VAR (* inputs/outputs *)

	ResetOld : BOOL;
	KeyResetOld : BOOL;
	AuxResetActivation : BOOL;
	ResetActivation : BOOL;
	Signals : ARRAY[1..256] OF BOOL;		(*each cell represents a signal code, used to know if signal is Active *)
	NumberOfAlarms : INT;			(* Counting processed alarms *)
	NumberOfAnomalies : INT;		(* Counting processed anomalies *)
	NumberOfWarnings : INT;		(* Counting processed warnings *)
	NumberOfInformation : INT;		(* Counting processed information *)
	ActiveSignalCodes : ARRAY[0..256] OF WORD;	(*each cell represents a Counted Active Signal Code, used to distinguish active/inactive in cronological sense*)
	NumberOfActiveAlarms : INT;		(* Counting active alarms *)
	NumberOfActiveAnomalies : INT;		(* Counting active anomalies *)
	NumberOfActiveWarning : INT;		(* Counting active warnings *)
	NumberOfActiveInformation : INT;	(* Counting active information *)
	SignalManagementError : BOOL;		(* not used for now *)
	Index : INT;	                             (*To trace working signal *)
	BaseIndex : INT;			(* To Trace offset depending on signal type *)
	i: INT;		(* Used in Reset Activation FOR Cycle *)
	AutoResetCondition: BOOL;	(* FALSE for Alarms/Anomalies, TRUE for Warning/Info *)
	AuxResetCondition: BOOL;	(* FALSE when AUX_RESET needed, TRUE for others *)
	SignalsCounters : ARRAY [1..256] OF INT;	(* Counters for Provisional Reset Condition *)
	ProvisionFlag: BOOL := FALSE;

END_VAR
CASE OperationType OF

	INIT: (* INIT PHASE *)			(* Reset Arrays - 1 Time*)

		IF KeyReset THEN

			FOR i:=1 TO 256 DO
				Signals[i] := FALSE;
				ActiveSignalCodes[i] := 0;		(* =NONE *)
				SignalsCounters[i] := 0;
			END_FOR

		END_IF

	START_CONFIGURATION: (* START_CONFIGURATION *)			(* Reset Alarms Count 1-Time *)

		NumberOfAlarms := 0;
		NumberOfAnomalies := 0;
		NumberOfWarnings := 0;
		NumberOfInformation := 0;

	CONFIGURATION:  (* CONFIGURATION PHASE*)					(* counting signals - Cycle over all possible signals *)

		CASE (WORD_TO_INT(SignalType AND SIGNAL_TYPE_MASK)) OF
			1:   (*ALARMS*)

				NumberOfAlarms := NumberOfAlarms + 1;

			2:   (*ANOMALIES*)

				NumberOfAnomalies := NumberOfAnomalies + 1;

			3:  (*WARNINGS*)

				NumberOfWarnings := NumberOfWarnings + 1;

			4:  (*INFORMATIONS*)

				NumberOfInformation := NumberOfInformation + 1;

		END_CASE

	START_GENERATION:  (* START GENERATION PHASE*)			(* Prepare for generation 1-Time *)

		ResetEnable := FALSE;
		AuxResetEnable := FALSE;
		SignalOutputs := NONE;

		ResetActivation := ResetSignal AND NOT ResetOld;		(* Set ResetActivation if Ext_Reset active *)
		ResetOld := Reset;		(*updateOLD*)

		AuxResetActivation := KeyReset (*AND NOT KeyResetOld*);   (* Not used Anymore... *)		(* Set AuxResetActivation if KeyReset Active*)
		(* KeyResetOld:= KeyReset;			(*updateOLD*) *)

	GENERATION: (* GENERATION PHASE *)

		AuxResetCondition := TRUE;
		ProvisionFlag := FALSE;

(*  Update, Index, Base Index and Condition : Cyclic*)

		CASE (SignalType AND SIGNAL_TYPE_MASK) OF

			1:
				Index := NumberOfActiveAlarms;
				BaseIndex := 0;
				AutoResetCondition := FALSE;
			2:
				Index := NumberOfActiveAnomalies;
				BaseIndex := NumberOfAlarms;
				AutoResetCondition := FALSE;
			3:
				Index := NumberOfActiveWarning;
				BaseIndex := NumberOfAlarms + NumberOfAnomalies;
				AutoResetCondition := TRUE;
			4:
				Index := NumberOfActiveInformation;
				BaseIndex := NumberOfAlarms + NumberOfAnomalies + NumberOfWarnings;
				AutoResetCondition := TRUE;
		END_CASE

(* Set AutoResetCondition if AUTO_RESET/.../... actives *)

		IF ((SignalType AND AUTO_RESET) = AUTO_RESET) THEN AutoResetCondition:=TRUE; END_IF
		IF ((SignalType AND AUTO_CONDITIONED_RESET) = AUTO_CONDITIONED_RESET)  AND AutoResetSignal THEN AutoResetCondition:=TRUE; END_IF
		IF ((SignalType AND UNCONDITIONED_RESET) = UNCONDITIONED_RESET) THEN AutoResetCondition:=TRUE; ActivationSignal:=FALSE; END_IF
		IF ((SignalType AND AUX_RESET) = AUX_RESET) THEN
			IF NOT AuxResetActivation THEN
				AuxResetCondition := FALSE;
			ELSE
				AutoResetCondition := TRUE;
			END_IF
		END_IF
		IF ((SignalType AND AUTO_PROVISIONAL_RESET) = AUTO_PROVISIONAL_RESET)  THEN
			IF ActivationSignal THEN
				IF  (SignalsCounters[SignalCode] > 0) THEN	(* timer not Expired, fake deactivation *)
					SignalsCounters[SignalCode] := SignalsCounters[SignalCode] - 1;
					ProvisionFlag := TRUE;
				END_IF
			ELSE
				SignalsCounters[SignalCode] := ProvisionalDelay;	(* Signal not active, update signal Timer *)
			END_IF
		END_IF

(* Activate Signal if ActivationSignalTRUE and not already activated *)

		IF ActivationSignal AND NOT Signals[SignalCode]  AND NOT ProvisionFlag THEN
			Signals[SignalCode] := TRUE;
			Index := Index + 1;
			ActiveSignalCodes[BaseIndex + Index] := SignalCode;
		END_IF
		IF AutoResetCondition AND Signals[SignalCode] AND NOT ActivationSignal AND (ActiveSignalCodes[BaseIndex + 1] = SignalCode) THEN 	(* Enable Reset if most important fault is not present anymore *)
			ResetEnable := TRUE;
			IF ((SignalCode AND AUX_RESET) = AUX_RESET) THEN AuxResetEnable:=TRUE; END_IF
		END_IF

(*Reset Most Important fault IF not present anymore and Reset Activated *)

		IF (ResetActivation OR AutoResetCondition) AND Signals[SignalCode] AND NOT ActivationSignal AND (ActiveSignalCodes[BaseIndex + 1] = SignalCode) AND  AuxResetCondition THEN

			Signals[SignalCode] := FALSE;

			FOR i := 2 TO Index DO
				ActiveSignalCodes[BaseIndex + i-1] := ActiveSignalCodes[BaseIndex + i];
			END_FOR;
			ActiveSignalCodes[BaseIndex + Index] := 0;
			Index := Index - 1;
			IF NOT CumulativeReset THEN ResetActivation := FALSE;	END_IF	(* COMMENT THIS LINE TO GO BACK TO CUMULATIVE RESET *)
		END_IF

(*  Update Number of Active Alarm or Anomaly or Warn or Info *)

	CASE (SignalType AND SIGNAL_TYPE_MASK) OF
			1:
				NumberOfActiveAlarms := Index;
			2:
				NumberOfActiveAnomalies := Index;
			3:
				NumberOfActiveWarning := Index;
			4:
				NumberOfActiveInformation := Index;
		END_CASE

(* Signal Priority Code (the one first in time), to prompt messages through bridgeCode2String *)

		IF (NumberOfActiveAlarms>0) THEN
			SignalPriorityCode := ActiveSignalCodes[1];
		ELSE
			IF (NumberOfActiveAnomalies>0) THEN
				SignalPriorityCode := ActiveSignalCodes[NumberOfAlarms+1];
			ELSE
				IF (NumberOfActiveWarning>0) THEN
					SignalPriorityCode := ActiveSignalCodes[NumberOfAlarms+NumberOfAnomalies+1];
				ELSE
					IF (NumberOfActiveInformation>0) THEN
						SignalPriorityCode := ActiveSignalCodes[NumberOfAlarms+NumberOfAnomalies+NumberOfWarnings+1];
					ELSE
						SignalPriorityCode := ActiveSignalCodes[0];
					END_IF
				END_IF
			END_IF
		END_IF

(* IF Signal is Active then Update Output *)

		IF Signals[SignalCode] THEN

			SignalOutputs := SignalOutputs OR SignalOutput;	(* old values + actual one *)

		END_IF

END_CASE
END_FUNCTION_BLOCK

(* POU MyLibraries/PrioritySignalToString, ST *)
FUNCTION PrioritySignalToString : STRING

VAR_INPUT

	SignalPriorityCode : WORD;

END_VAR
CASE (WORD_TO_INT(SignalPriorityCode)) OF
  0:
      PrioritySignalToString := 'NONE';

  3:
      PrioritySignalToString := 'Emergency Button Pressed';

  4:
      PrioritySignalToString := 'Freeze Button Pressed';

  5:
      PrioritySignalToString := '(OnPhase)Stop Button Pressed';

  131:
      PrioritySignalToString := 'Machine Stopped for Inactivity ';

  191:
      PrioritySignalToString := 'S1.Info: Warehouse is Empty ';

  198:
      PrioritySignalToString := 'S4.Info: No Cover in AssemblyStation';

  21:
      PrioritySignalToString := 'S1.ActuatorFault: Cylinder ';

  23:
      PrioritySignalToString := 'S1.ActuatorFault: RotaryArm ';

  26:
      PrioritySignalToString := 'S1.ActuatorFault: Vacuum ';

  28:
      PrioritySignalToString := 'S1.ActuatorFault: ExpulsionAir ';

  31:
      PrioritySignalToString := 'S2.ActuatorFault: Elevator ';

  34:
      PrioritySignalToString := 'S2.ActuatorFault: Cylinder ';

  36:
      PrioritySignalToString := 'S2.ActuatorFault: AirSlider ';

  41:
      PrioritySignalToString := 'S3.ActuatorFault: Rotary Motor ';

  43:
      PrioritySignalToString := 'S3.ActuatorFault: Load Inspector ';

  45:
      PrioritySignalToString := 'S3.ActuatorFault: DrillCylinder ';

  47:
      PrioritySignalToString := 'S3.ActuatorFault: Driller ';

  48:
      PrioritySignalToString := 'S3.ActuatorFault: Blocker ';

  49:
      PrioritySignalToString := 'S3.ActuatorFault: Expeller ';

  51:
      PrioritySignalToString := 'S4.ActuatorFault: SpringExtractor ';

  52:
      PrioritySignalToString := 'S4.ActuatorFault: PistonSelector ';

  53:
      PrioritySignalToString := 'S4.ActuatorFault: CoverExtractor ';

  54:
      PrioritySignalToString := 'S4.RobotFault: LoadBlocker ';

  56:
      PrioritySignalToString := 'S4.RobotFault: InitActuation ';

  57:
      PrioritySignalToString := 'S4.RobotFault: PistonActuation';

  58:
      PrioritySignalToString := 'S4.RobotFault: SpringActuation ';

  59:
      PrioritySignalToString := 'S4.RobotFault: CoverActuation ';

  60:
      PrioritySignalToString := 'S4.RobotFault: AssemblyActuation ';



  81:
      PrioritySignalToString := 'S1.SensorFault: Cylinder ';

  84:
      PrioritySignalToString := 'S1.SensorFault: RotaryArm ';

  87:
      PrioritySignalToString := 'S1.SensorFault: Vacuum ';

  91:
      PrioritySignalToString := 'S2.SensorFault: Elevator ';

  94:
      PrioritySignalToString := 'S2.SensorFault: Cylinder ';

  101:
      PrioritySignalToString := 'S3.SensorFault: RotaryAlignment ';

  103:
      PrioritySignalToString := 'S3.SensorFault: DrillCylinder ';

  111:
      PrioritySignalToString := 'S4.SensorFault: SpringExtractor ';

  112:
      PrioritySignalToString := 'S4.SensorFault: PistonSelector ';

  113:
      PrioritySignalToString := 'S4.SensorFault: CoverExtractor ';

  115:
      PrioritySignalToString := 'S4.RobotFault: InitSensor ';

  116:
      PrioritySignalToString := 'S4.RobotFault: PistonSensorr ';

  117:
      PrioritySignalToString := 'S4.RobotFault: SpringSensor ';

  118:
      PrioritySignalToString := 'S4.RobotFault: CoverSensor ';

  119:
      PrioritySignalToString := 'S4.RobotFault: AssemblySensor ';

END_CASE
END_FUNCTION

(* POU Bridge/OutputBridge, ST *)
PROGRAM OutputBridge
VAR

END_VAR
(*Actuation of the 1° station*)

CylinderExtractsLoadFromWarehouse :=  FaultSim(FaultLow:= CylinderExtractsLoadFromWarehouseBlock , FaultHigh := CylinderExtractsLoadFromWarehouseBlockHigh , Input := A_Cylinder1);
RotaryMakerVsWarehouse :=  FaultSim(FaultLow:= RotaryMakerVsWarehouseBlock , FaultHigh := RotaryMakerVsWarehouseBlockHigh , Input := A_ArmToWarehouse1);
RotaryMakerVsVerification :=  FaultSim(FaultLow:= RotaryMakerVsVerificationBlock , FaultHigh := RotaryMakerVsVerificationBlockHigh , Input := A_ArmToElevator1);
VacuumGenerator :=  FaultSim(FaultLow:= VacuumGeneratorBlock , FaultHigh := VacuumGeneratorBlockHigh , Input := A_Vacuum1);
ExpulsionAirVacuum :=  FaultSim(FaultLow:= ExpulsionAirVacuumBlock , FaultHigh := ExpulsionAirVacuumBlockHigh , Input := A_AirVacuum1);

(*Actuation of the 2° station*)

ToLiftCylinderToMeasureLoad :=  FaultSim(FaultLow:= ToLiftCylinderToMeasureLoadBlock , FaultHigh := ToLiftCylinderToMeasureLoadBlockHigh , Input := A_ElevatorUp2);
ToLowerCylinderToMeasureLoad :=  FaultSim(FaultLow:= ToLowerCylinderToMeasureLoadBlock , FaultHigh := ToLiftCylinderToMeasureLoadBlockHigh , Input := A_ElevatorDown2);
ToExtendCylinderOfExtractionVsGuide :=  FaultSim(FaultLow:= ToExtendCylinderOfExtractionVsGuideBlock , FaultHigh := ToExtendCylinderOfExtractionVsGuideBlockHigh , Input := A_Cylinder2);
AirCushion :=  FaultSim(FaultLow:= AirCushionBlock , FaultHigh := AirCushionBlockHigh , Input := A_AirSlider2);
AirCushion :=  FaultSim(FaultLow:= AirCushionBlock , FaultHigh := AirCushionBlockHigh , Input := A_AirSlider2);
UncorrectComparison := L_PieceToDiscard2;

(*Actuation of the 3° station*)

RotaryTableMotor :=  FaultSim(FaultLow:= RotaryTableMotorBlockLow , FaultHigh := RotaryTableMotorBlockHigh , Input := A_RotaryTable3);
ToLowerCylinderToInspectLoad :=  FaultSim(FaultLow:= ToLowerCylinderToInspectLoadBlockLow , FaultHigh := ToLowerCylinderToInspectLoadBlockHigh , Input := A_GoControl3);
ToLiftDrillingUnit :=  FaultSim(FaultLow:= ToLiftDrillingUnitBlockLow , FaultHigh := ToLiftDrillingUnitBlockHigh , Input := A_ReturnDrill3);
ToLowerDrillingUnit :=  FaultSim(FaultLow:= ToLowerDrillingUnitBlockLow , FaultHigh := ToLowerDrillingUnitBlockHigh , Input :=A_GoDrill3 );
DrillingUnitActive :=  FaultSim(FaultLow:= DrillingUnitActiveBlockLow , FaultHigh := DrillingUnitActiveBlockHigh , Input :=A_Drilling3);
BlockingCylinderForwardInDrillingPositioning :=  FaultSim(FaultLow:= BlockingCylinderForwardInDrillingPositioningBlockLow , FaultHigh := BlockingCylinderForwardInDrillingPositioningBlockHigh , Input := A_BlockElement3);
ExpellingLeverActive :=  FaultSim(FaultLow:= ExpellingLeverActiveBlockLow , FaultHigh := ExpellingLeverActiveBlockHigh , Input := A_ExpellElement3);

(*Actuation of the 4° station*)

ToExtractSpringInAssemblyStation :=  FaultSim(FaultLow:= ToExtractSpringInAssemblyStationBlockLow , FaultHigh := ToExtractSpringInAssemblyStationBlockHigh , Input := A_SpringCylinder4);
PistonSelectorGoOnTheRight :=  FaultSim(FaultLow:= PistonSelectorGoOnTheRightBlockLow , FaultHigh := PistonSelectorGoOnTheRightBlockHigh , Input := A_GiveBlackPiston4);
PistonSelectorGoOnTheLeft :=  FaultSim(FaultLow:= PistonSelectorGoOnTheLeftBlockLow , FaultHigh := PistonSelectorGoOnTheLeftBlockHigh , Input := A_GiveSilverPiston4);
ToExtractCoverInAssemblyStationForward :=  FaultSim(FaultLow:= ToExtractCoverInAssemblyStationForwardBlockLow , FaultHigh := ToExtractCoverInAssemblyStationForwardBlockHigh , Input := A_CoverCylinder4);
BlockingCylinderForwardInAssemblyStation :=  FaultSim(FaultLow:= BlockingCylinderForwardInAssemblyStationBlockLow , FaultHigh := BlockingCylinderForwardInAssemblyStationBlockHigh , Input := A_BlockElement4);

(*Robot actuation*)

RobotGoToInitialPosition :=  FaultSim(FaultLow:= RobotGoToInitialPositionBlockLow , FaultHigh := RobotGoToInitialPositionBlockHigh , Input := A_RobotToInitial4);
RobotTakeBlackLoad :=  FaultSim(FaultLow:= RobotTakeBlackLoadBlockLow , FaultHigh := RobotTakeBlackLoadBlockHigh , Input := A_RobotTakeBlack4);
RobotTakeRedSilverLoad :=  FaultSim(FaultLow:= RobotTakeRedSilverLoadBlockLow , FaultHigh := RobotTakeRedSilverLoadBlockHigh , Input := A_RobotTakeRedSilver4);
RobotTakeLoadToDiascardBlack :=  FaultSim(FaultLow:= RobotTakeLoadToDiascardBlockLow , FaultHigh := RobotTakeLoadToDiascardBlockHigh , Input := A_RobotDiscardBlack4);
RobotTakeLoadToDiascardRedSilver :=  FaultSim(FaultLow:= RobotTakeLoadToDiascardBlockLow , FaultHigh := RobotTakeLoadToDiascardBlockHigh , Input := A_RobotDiscardRedSilver4);
RobotTakeCurrentLoadToAssembly :=  FaultSim(FaultLow:= RobotTakeCurrentLoadToAssemblyBlockLow , FaultHigh := RobotTakeCurrentLoadToAssemblyBlockHigh , Input := A_RobotAssembly4);
RobotGoToPistonHouse :=  FaultSim(FaultLow:= RobotGoToPistonHouseBlockLow , FaultHigh := RobotGoToPistonHouseBlockHigh , Input := A_RobotPiston4);
RobotGoToSpringHouse :=  FaultSim(FaultLow:= RobotGoToSpringHouseBlockLow , FaultHigh := RobotGoToSpringHouseBlockHigh , Input := A_RobotSpring4);
RobotGoToCoverHouse :=  FaultSim(FaultLow:= RobotGoToCoverHouseBlockLow , FaultHigh := RobotGoToCoverHouseBlockHigh , Input := A_RobotCover4);
RobotReset := A_RobotReset4;

(*Simulation of robot actuators*)

IF RobotGoToInitialPosition THEN
	Bit3Output := FALSE;
	Bit2Output := FALSE;
	Bit1Output := FALSE;
	Bit0Output := TRUE;
END_IF

IF RobotTakeBlackLoad THEN
	Bit3Output := FALSE;
	Bit2Output := FALSE;
	Bit1Output := TRUE;
	Bit0Output := FALSE;
END_IF

IF RobotTakeRedSilverLoad THEN
	Bit3Output := FALSE;
	Bit2Output := FALSE;
	Bit1Output := TRUE;
	Bit0Output := TRUE;
END_IF

IF RobotTakeLoadToDiascardBlack THEN
	Bit3Output := FALSE;
	Bit2Output := TRUE;
	Bit1Output := FALSE;
	Bit0Output := TRUE;
END_IF

IF RobotTakeLoadToDiascardRedSilver THEN
	Bit3Output := FALSE;
	Bit2Output := TRUE;
	Bit1Output := FALSE;
	Bit0Output := FALSE;
END_IF

IF RobotTakeCurrentLoadToAssembly THEN
	Bit3Output := TRUE;
	Bit2Output := FALSE;
	Bit1Output := FALSE;
	Bit0Output := TRUE;
END_IF

IF RobotGoToPistonHouse THEN
	Bit3Output := FALSE;
	Bit2Output := TRUE;
	Bit1Output := TRUE;
	Bit0Output := TRUE;
END_IF

IF RobotGoToSpringHouse THEN
	Bit3Output := FALSE;
	Bit2Output := TRUE;
	Bit1Output := TRUE;
	Bit0Output := FALSE;
END_IF

IF RobotGoToCoverHouse THEN
	Bit3Output := TRUE;
	Bit2Output := FALSE;
	Bit1Output := FALSE;
	Bit0Output := FALSE;
END_IF

IF RobotReset THEN
	Bit3Output := FALSE;
	Bit2Output := FALSE;
	Bit1Output := FALSE;
	Bit0Output := FALSE;
END_IF

Bit4Output := StopOutput4;

(*Lights*)

LightStart := L_Start;
LightReset := L_Reset;
LightEmptyWarehouse := L_EmptyWarehouse;
LightUpsideDownLoadInExpelling := L_UpsideDownElement;
LightEmptyCoverHouse := L_NoCover;
LightRobotInMovement := L_RobotMoving;
LightRobotServoON := L_RobotOn;
LightRedLoad := L_RedSilverElement;
LightBlackLoad := L_BlackElement;


(*General State Machine*)

IndicatorStateInit:=VL_StateInit;
IndicatorStateReady:=VL_StateReady;
IndicatorStateRun:=VL_StateRun;
IndicatorStateAlarm:=VL_StateAlarm;
IndicatorStateFreeze:=VL_StateImmediateStop;
IndicatorStateStop:=VL_StateStop;
IndicatorStateReset:=VL_StateReset;

(*Virtual panel variable*)

ColorVisualization[2]:=VL_ColorVis2;
ColorVisualization[3] := VL_ColorVis;
PositionVisualization[3] := VL_PositionVis;
ColorVisualization[4] := VL_ColorVis4;
ElementCompleted4 := VL_Completed;
ElementRejected4:=VL_Rejected;
END_PROGRAM

(* POU MyLibraries/Filter, ST *)
(* @OBJECTFLAGS := '0, 8' *)
FUNCTIONBLOCK Filter

VAR_INPUT

	OperationType : INT;
	Clock : BOOL;
	Signal : BOOL;
	ActivationDelay : UDINT;
	DeactivationDelay : UDINT;

END_VAR

VAR_OUTPUT

	DelayedSignal : BOOL;

END_VAR

VAR

	Delay : UDINT;

END_VAR
IF (OperationType = INIT) THEN
	Delay := 0;
ELSE
	IF (Signal = DelayedSignal) THEN
		IF (Signal) THEN
			Delay := DeactivationDelay;
		ELSE
			Delay := ActivationDelay;
		END_IF
	END_IF
END_IF

IF (Clock AND (Delay > 0)) THEN
	Delay := Delay - 1;
END_IF

IF (Delay = 0) THEN
	DelayedSignal := Signal;
END_IF
END_FUNCTION_BLOCK

(* Visualisation Fault_Detection
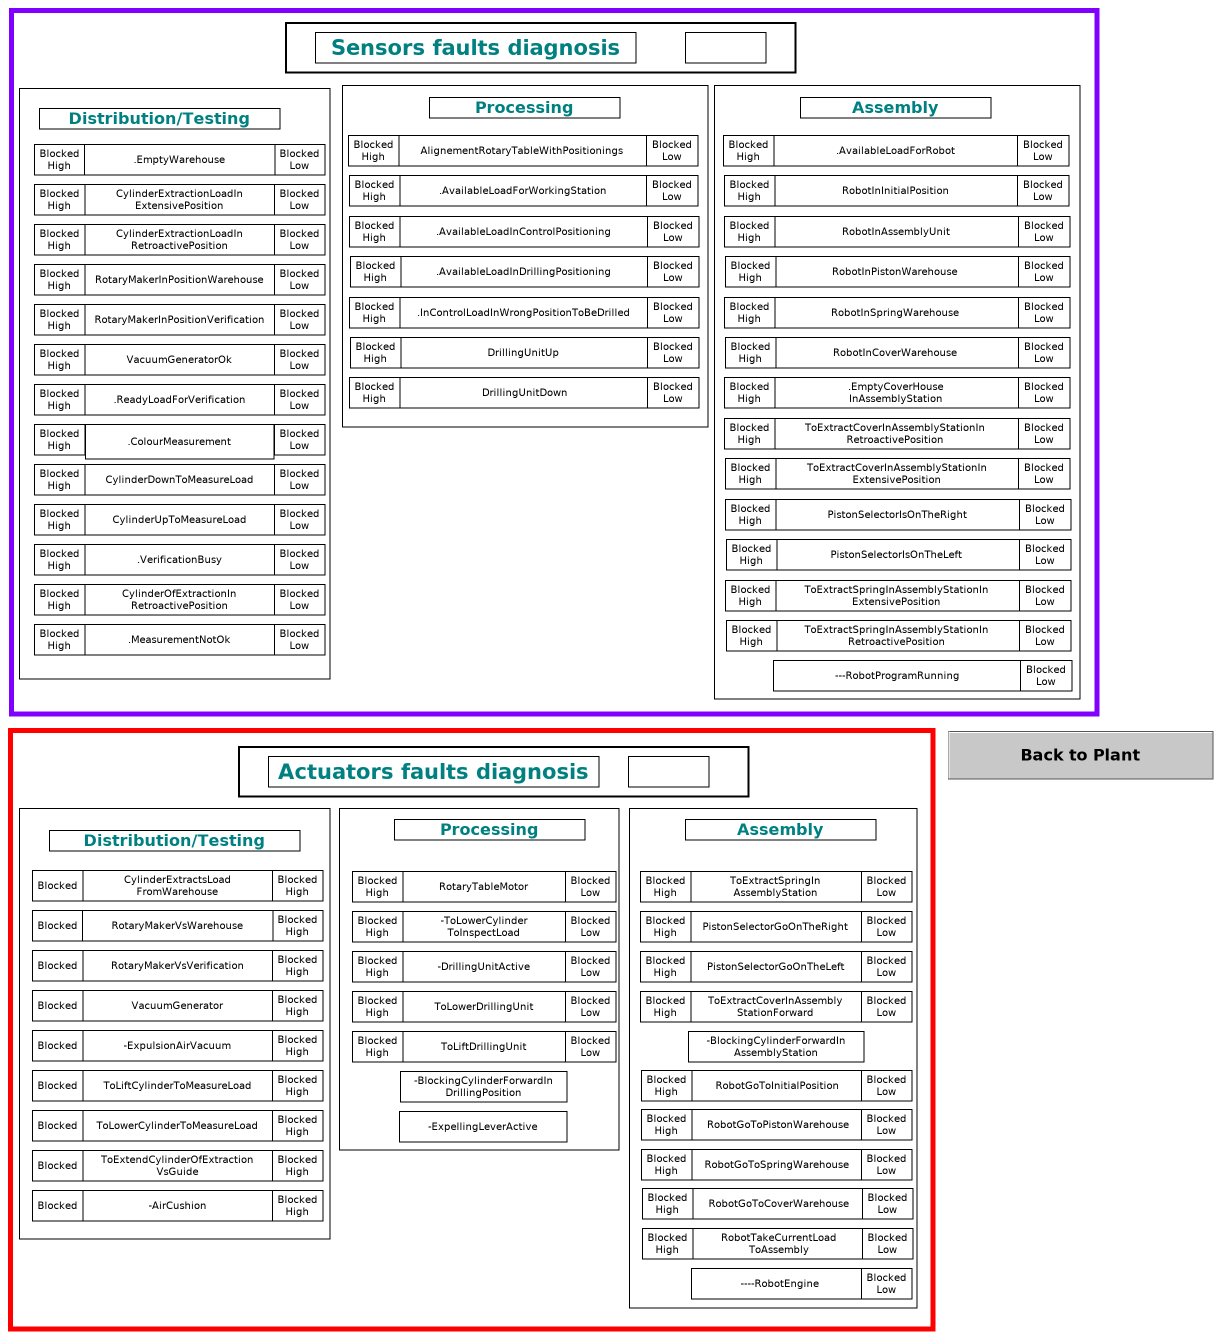
rounded rectangle at (316,34)-(637,65): text "Sensors faults diagnosis"
rounded rectangle at (269,758)-(600,789): text "Actuators faults diagnosis"
button at (949,733)-(1214,781): text "Back to Plant"; opens FESTO_Interface
rectangle at (40,110)-(281,131): text "Distribution/Testing"
rectangle at (35,146)-(86,177): text "Blocked / High"; alarm colour if EmptyWarehouseBlockedHigh
rectangle at (275,146)-(326,177): text "Blocked / Low"; alarm colour if EmptyWarehouseBlockedLow
rectangle at (85,146)-(276,177): text ".EmptyWarehouse"; alarm colour if EmptyWarehouseBlockedHigh OR EmptyWarehouseBlockedLow
rectangle at (85,186)-(276,217): text "CylinderExtractionLoadIn / ExtensivePosition"; alarm colour if F_S_Cylinder1
rectangle at (85,226)-(276,257): text "CylinderExtractionLoadIn / RetroactivePosition"; alarm colour if F_S_Cylinder1
rectangle at (85,266)-(276,297): text "RotaryMakerInPositionWarehouse"; alarm colour if F_S_Rotary1
rectangle at (85,306)-(276,337): text "RotaryMakerInPositionVerification"; alarm colour if F_S_Rotary1
rectangle at (85,346)-(276,377): text "VacuumGeneratorOk"; alarm colour if F_S_Vacuum1
rectangle at (85,386)-(276,417): text ".ReadyLoadForVerification"; alarm colour if ReadyLoadForVerificationBlockedHigh OR ReadyLoadForVerificationBlockedLow
rectangle at (86,426)-(275,461): text ".ColourMeasurement"; alarm colour if ColourMeasurementBlockedHigh OR ColourMeasurementBlockedLow
rectangle at (85,466)-(276,497): text "CylinderDownToMeasureLoad"; alarm colour if F_S_Elevator2
rectangle at (85,506)-(276,537): text "CylinderUpToMeasureLoad"; alarm colour if F_S_Elevator2
rectangle at (85,546)-(276,577): text ".VerificationBusy"; alarm colour if VerificationBusyBlockedHigh OR VerificationBusyBlockedLow
rectangle at (85,586)-(276,617): text "CylinderOfExtractionIn / RetroactivePosition"; alarm colour if F_S_Cylinder2
rectangle at (85,626)-(276,657): text ".MeasurementNotOk"
rectangle at (35,186)-(86,217): text "Blocked / High"; alarm colour if FH_ES_Cylinder1
rectangle at (275,186)-(326,217): text "Blocked / Low"; alarm colour if FL_ES_Cylinder1
rectangle at (35,226)-(86,257): text "Blocked / High"; alarm colour if FH_DS_Cylinder1
rectangle at (275,226)-(326,257): text "Blocked / Low"; alarm colour if FL_DS_Cylinder1
rectangle at (35,266)-(86,297): text "Blocked / High"; alarm colour if FH_ES_Rotary1
rectangle at (275,266)-(326,297): text "Blocked / Low"; alarm colour if FL_ES_Rotary1
rectangle at (35,306)-(86,337): text "Blocked / High"; alarm colour if FH_DS_Rotary1
rectangle at (275,306)-(326,337): text "Blocked / Low"; alarm colour if FL_DS_Rotary1
rectangle at (35,346)-(86,377): text "Blocked / High"; alarm colour if FH_S_Vacuum1
rectangle at (275,346)-(326,377): text "Blocked / Low"; alarm colour if FL_S_Vacuum1
rectangle at (35,386)-(86,417): text "Blocked / High"; alarm colour if ReadyLoadForVerificationBlockedHigh
rectangle at (275,386)-(326,417): text "Blocked / Low"; alarm colour if ReadyLoadForVerificationBlockedLow
rectangle at (35,426)-(86,457): text "Blocked / High"; alarm colour if ColourMeasurementBlockedHigh
rectangle at (275,426)-(326,457): text "Blocked / Low"; alarm colour if ColourMeasurementBlockedLow
rectangle at (35,466)-(86,497): text "Blocked / High"; alarm colour if FH_DS_Elevator2
rectangle at (275,466)-(326,497): text "Blocked / Low"; alarm colour if FL_DS_Elevator2
rectangle at (35,506)-(86,537): text "Blocked / High"; alarm colour if FH_ES_Elevator2
rectangle at (275,506)-(326,537): text "Blocked / Low"; alarm colour if FL_ES_Elevator2
rectangle at (35,546)-(86,577): text "Blocked / High"; alarm colour if VerificationBusyBlockedHigh
rectangle at (275,546)-(326,577): text "Blocked / Low"; alarm colour if VerificationBusyBlockedLow
rectangle at (35,586)-(86,617): text "Blocked / High"; alarm colour if FH_S_Cylinder2
rectangle at (275,586)-(326,617): text "Blocked / Low"; alarm colour if FL_S_Cylinder2
rectangle at (35,626)-(86,657): text "Blocked / High"; alarm colour if MeasurementNotOkBlockedHigh
rectangle at (275,626)-(326,657): text "Blocked / Low"; alarm colour if MeasurementNotOkBlockedLow
rectangle at (50,832)-(301,853): text "Distribution/Testing"
rectangle at (83,872)-(274,903): text "CylinderExtractsLoad / FromWarehouse"; alarm colour if F_A_Cylinder1
rectangle at (83,952)-(274,983): text "RotaryMakerVsVerification"; alarm colour if F_A_Rotary1
rectangle at (83,992)-(274,1023): text "VacuumGenerator"; alarm colour if F_A_Vacuum1
rectangle at (83,1032)-(274,1063): text "-ExpulsionAirVacuum"; alarm colour if ExpulsionAirVacuumBlocked OR ExpulsionAirVacuumBlockedHigh
rectangle at (83,1072)-(274,1103): text "ToLiftCylinderToMeasureLoad"; alarm colour if F_A_Elevator2
rectangle at (83,1112)-(274,1143): text "ToLowerCylinderToMeasureLoad"; alarm colour if F_A_Elevator2
rectangle at (83,1192)-(274,1223): text "-AirCushion"; alarm colour if AirCushionBlocked OR AirCushionBlockedHigh
rectangle at (83,1152)-(274,1183): text "ToExtendCylinderOfExtraction / VsGuide"; alarm colour if F_A_Cylinder2
rectangle at (273,872)-(324,903): text "Blocked / High"; alarm colour if FH_A_Cylinder1
rectangle at (273,912)-(324,943): text "Blocked / High"; alarm colour if FH_EA_Rotary1
rectangle at (273,952)-(324,983): text "Blocked / High"; alarm colour if FH_DA_Rotary1
rectangle at (273,992)-(324,1023): text "Blocked / High"; alarm colour if FH_A_Vacuum1
rectangle at (273,1032)-(324,1063): text "Blocked / High"; alarm colour if FH_A_Expulsion1
rectangle at (273,1072)-(324,1103): text "Blocked / High"; alarm colour if FH_EA_Elevator2
rectangle at (273,1112)-(324,1143): text "Blocked / High"; alarm colour if FH_DA_Elevator2
rectangle at (273,1152)-(324,1183): text "Blocked / High"; alarm colour if FH_A_Cylinder2
rectangle at (273,1192)-(324,1223): text "Blocked / High"; alarm colour if FH_A_Air2
rectangle at (33,872)-(84,903): text "Blocked"; alarm colour if FL_A_Cylinder1
rectangle at (33,912)-(84,943): text "Blocked"; alarm colour if FL_EA_Rotary1
rectangle at (33,952)-(84,983): text "Blocked"; alarm colour if FL_DA_Rotary1
rectangle at (33,992)-(84,1023): text "Blocked"; alarm colour if FL_A_Vacuum1
rectangle at (33,1032)-(84,1063): text "Blocked"; alarm colour if FL_A_Expulsion1
rectangle at (33,1072)-(84,1103): text "Blocked"; alarm colour if FL_EA_Elevator2
rectangle at (33,1112)-(84,1143): text "Blocked"; alarm colour if FL_DA_Elevator2
rectangle at (33,1152)-(84,1183): text "Blocked"; alarm colour if FL_A_Cylinder2
rectangle at (33,1192)-(84,1223): text "Blocked"; alarm colour if FL_A_Air2
rectangle at (83,912)-(274,943): text "RotaryMakerVsWarehouse"; alarm colour if F_A_Rotary1
rectangle at (430,99)-(621,120): text "Processing"
rectangle at (801,99)-(992,120): text "Assembly"
rectangle at (397,137)-(649,168): text "AlignementRotaryTableWithPositionings"; alarm colour if F_S_RotaryTable3
rectangle at (399,177)-(649,208): text ".AvailableLoadForWorkingStation"
rectangle at (399,218)-(650,249): text ".AvailableLoadInControlPositioning"
rectangle at (399,258)-(650,289): text ".AvailableLoadInDrillingPositioning"
rectangle at (399,299)-(650,330): text ".InControlLoadInWrongPositionToBeDrilled"
rectangle at (399,339)-(650,370): text "DrillingUnitUp"; alarm colour if F_S_DrillCylinder3
rectangle at (399,379)-(653,410): text "DrillingUnitDown"; alarm colour if F_S_DrillCylinder3
rectangle at (773,137)-(1020,168): text ".AvailableLoadForRobot"
rectangle at (773,177)-(1020,208): text "RobotInInitialPosition"; alarm colour if F_S_RobotInInitial4
rectangle at (773,218)-(1021,249): text "RobotInAssemblyUnit"; alarm colour if F_S_RobotAssembly4
rectangle at (771,258)-(1021,289): text "RobotInPistonWarehouse"; alarm colour if F_S_RobotPiston4
rectangle at (771,299)-(1021,330): text "RobotInSpringWarehouse"; alarm colour if F_S_RobotSpring4
rectangle at (771,339)-(1021,370): text "RobotInCoverWarehouse"; alarm colour if F_S_RobotCover4
rectangle at (771,379)-(1023,410): text ".EmptyCoverHouse / InAssemblyStation"
rectangle at (771,420)-(1021,451): text "ToExtractCoverInAssemblyStationIn / RetroactivePosition"; alarm colour if F_S_ExtractCover4
rectangle at (775,460)-(1021,491): text "ToExtractCoverInAssemblyStationIn / ExtensivePosition"; alarm colour if F_S_ExtractCover4
rectangle at (775,501)-(1022,532): text "PistonSelectorIsOnTheRight"; alarm colour if F_S_PistonSelector4
rectangle at (773,541)-(1022,572): text "PistonSelectorIsOnTheLeft"; alarm colour if F_S_PistonSelector4
rectangle at (773,582)-(1022,613): text "ToExtractSpringInAssemblyStationIn / ExtensivePosition"; alarm colour if F_S_SpringExtractor4
rectangle at (773,622)-(1022,653): text "ToExtractSpringInAssemblyStationIn / RetroactivePosition"; alarm colour if F_S_SpringExtractor4
rectangle at (1018,137)-(1070,168): text "Blocked / Low"; alarm colour if AvailableLoadForRobotBlockedLow
rectangle at (1018,177)-(1070,208): text "Blocked / Low"; alarm colour if RobotInInitialPositionBlockedLow
rectangle at (1019,218)-(1071,249): text "Blocked / Low"; alarm colour if RobotInAssemblyUnitBlockedLow
rectangle at (1019,258)-(1071,289): text "Blocked / Low"; alarm colour if RobotInPistonWarehouseBlockedLow
rectangle at (1019,299)-(1071,330): text "Blocked / Low"; alarm colour if RobotInSpringWarehouseBlockedLow
rectangle at (1019,339)-(1071,370): text "Blocked / Low"; alarm colour if RobotInCoverWarehouseBlockedLow
rectangle at (1019,379)-(1071,410): text "Blocked / Low"; alarm colour if EmptyCoverHouseInAssemblyStationBlockedLow
rectangle at (1019,420)-(1071,451): text "Blocked / Low"; alarm colour if FL_DS_ExtractCover4
rectangle at (1019,460)-(1071,491): text "Blocked / Low"; alarm colour if FL_ES_ExtractCover4
rectangle at (1020,501)-(1072,532): text "Blocked / Low"; alarm colour if FL_ES_PistonSelector4
rectangle at (1020,541)-(1072,572): text "Blocked / Low"; alarm colour if FH_DS_PistonSelector4
rectangle at (1020,582)-(1072,613): text "Blocked / Low"; alarm colour if FL_ES_SpringExtractor4
rectangle at (1020,622)-(1072,653): text "Blocked / Low"; alarm colour if FL_DS_SpringExtractor4
rectangle at (724,137)-(775,168): text "Blocked / High"; alarm colour if AvailableLoadForRobotBlockedHigh
rectangle at (725,177)-(776,208): text "Blocked / High"; alarm colour if RobotInInitialPositionBlockedHigh
rectangle at (725,218)-(776,249): text "Blocked / High"; alarm colour if RobotInAssemblyUnitBlockedHigh
rectangle at (726,258)-(777,289): text "Blocked / High"; alarm colour if RobotInPistonWarehouseBlockedHigh
rectangle at (725,299)-(776,330): text "Blocked / High"; alarm colour if RobotInSpringWarehouseBlockedHigh
rectangle at (726,339)-(777,370): text "Blocked / High"; alarm colour if RobotInCoverWarehouseBlockedHigh
rectangle at (725,379)-(776,410): text "Blocked / High"; alarm colour if EmptyCoverHouseInAssemblyStationBlockedHigh
rectangle at (725,420)-(776,451): text "Blocked / High"; alarm colour if FH_DS_ExtractCover4
rectangle at (726,460)-(777,491): text "Blocked / High"; alarm colour if FH_ES_ExtractCover4
rectangle at (726,501)-(777,532): text "Blocked / High"; alarm colour if FH_ES_PistonSelector4
rectangle at (727,541)-(778,572): text "Blocked / High"; alarm colour if FL_DS_PistonSelector4
rectangle at (726,582)-(777,613): text "Blocked / High"; alarm colour if FH_ES_SpringExtractor4
rectangle at (727,622)-(778,653): text "Blocked / High"; alarm colour if FH_DS_SpringExtractor4
rectangle at (647,137)-(699,168): text "Blocked / Low"; alarm colour if FL_S_RotaryTable3
rectangle at (647,177)-(699,208): text "Blocked / Low"; alarm colour if AvailableLoadForWorkingStationBlockedLow
rectangle at (648,218)-(700,249): text "Blocked / Low"; alarm colour if AvailableLoadInControlPositioningBlockedLow
rectangle at (648,258)-(700,289): text "Blocked / Low"; alarm colour if AvailableLoadInDrillingPositioningBlockedLow
rectangle at (648,299)-(700,330): text "Blocked / Low"; alarm colour if InControlLoadInWrongPositionToBeDrilledBlockedLow
rectangle at (648,339)-(700,370): text "Blocked / Low"; alarm colour if FL_DS_DrillCylinder3
rectangle at (648,379)-(700,410): text "Blocked / Low"; alarm colour if FL_ES_DrillCylinder3
rectangle at (349,137)-(400,168): text "Blocked / High"; alarm colour if FH_S_RotaryTable3
rectangle at (350,177)-(401,208): text "Blocked / High"; alarm colour if AvailableLoadForWorkingStationBlockedHigh
rectangle at (350,218)-(401,249): text "Blocked / High"; alarm colour if AvailableLoadInControlPositioningBlockedHigh
rectangle at (351,258)-(402,289): text "Blocked / High"; alarm colour if AvailableLoadInDrillingPositioningBlockedHigh
rectangle at (350,299)-(401,330): text "Blocked / High"; alarm colour if InControlLoadInWrongPositionToBeDrilledBlockedHigh
rectangle at (351,339)-(402,370): text "Blocked / High"; alarm colour if FH_DS_DrillCylinder3
rectangle at (350,379)-(401,410): text "Blocked / High"; alarm colour if FH_ES_DrillCylinder3
rectangle at (774,662)-(1023,693): text "---RobotProgramRunning"
rectangle at (1021,662)-(1073,693): text "Blocked / Low"; alarm colour if RobotProgramRunningBlockedLow
rectangle at (395,821)-(586,842): text "Processing"
rectangle at (686,821)-(877,842): text "Assembly"
rectangle at (688,873)-(865,904): text "ToExtractSpringIn / AssemblyStation"; alarm colour if F_A_SpringExtractor4
rectangle at (688,913)-(865,944): text "PistonSelectorGoOnTheRight"; alarm colour if F_A_PistonSelector4
rectangle at (689,953)-(865,984): text "PistonSelectorGoOnTheLeft"; alarm colour if F_A_PistonSelector4
rectangle at (688,993)-(865,1024): text "ToExtractCoverInAssembly / StationForward"; alarm colour if F_A_ExtractCover4
rectangle at (689,1033)-(865,1064): text "-BlockingCylinderForwardIn / AssemblyStation"
rectangle at (688,1072)-(869,1103): text "RobotGoToInitialPosition"; alarm colour if F_A_RobotToInitial4
rectangle at (686,1151)-(870,1182): text "RobotGoToSpringWarehouse"; alarm colour if F_A_RobotSpring4
rectangle at (688,1111)-(870,1142): text "RobotGoToPistonWarehouse"; alarm colour if F_A_RobotPiston4
rectangle at (401,873)-(568,904): text "RotaryTableMotor"; alarm colour if F_A_RotaryTable3
rectangle at (402,913)-(568,944): text "-ToLowerCylinder / ToInspectLoad"
rectangle at (402,953)-(568,984): text "-DrillingUnitActive"
rectangle at (402,993)-(568,1024): text "ToLowerDrillingUnit"; alarm colour if F_A_DrillCylinder3
rectangle at (402,1033)-(568,1064): text "ToLiftDrillingUnit"; alarm colour if F_A_DrillCylinder3
rectangle at (400,1113)-(568,1144): text "-ExpellingLeverActive"
rectangle at (401,1073)-(568,1104): text "-BlockingCylinderForwardIn / DrillingPosition"
rectangle at (353,873)-(404,904): text "Blocked / High"; alarm colour if FH_A_RotaryTable3
rectangle at (353,913)-(404,944): text "Blocked / High"; alarm colour if FH_A_Cylinder3
rectangle at (353,953)-(404,984): text "Blocked / High"; alarm colour if FH_A_Drilling3
rectangle at (353,993)-(404,1024): text "Blocked / High"; alarm colour if FH_EA_DrillCylinder3
rectangle at (353,1033)-(404,1064): text "Blocked / High"; alarm colour if FH_DA_DrillCylinder3
rectangle at (566,873)-(617,904): text "Blocked / Low"; alarm colour if FL_A_RotaryTable3
rectangle at (566,913)-(617,944): text "Blocked / Low"; alarm colour if FL_A_Cylinder3
rectangle at (566,953)-(617,984): text "Blocked / Low"; alarm colour if FL_A_Drilling3
rectangle at (566,993)-(617,1024): text "Blocked / Low"; alarm colour if FL_EA_DrillCylinder3
rectangle at (566,1033)-(617,1064): text "Blocked / Low"; alarm colour if FL_DA_DrillCylinder3
rectangle at (641,873)-(692,904): text "Blocked / High"; alarm colour if FH_A_SpringExtractor4
rectangle at (641,913)-(692,944): text "Blocked / High"; alarm colour if FH_EA_PistonSelector4
rectangle at (641,953)-(692,984): text "Blocked / High"; alarm colour if FH_DA_PistonSelector4
rectangle at (641,993)-(692,1024): text "Blocked / High"; alarm colour if FH_A_ExtractCover4
rectangle at (862,873)-(913,904): text "Blocked / Low"; alarm colour if FL_A_SpringExtractor4
rectangle at (862,913)-(913,944): text "Blocked / Low"; alarm colour if FL_EA_PistonSelector4
rectangle at (862,953)-(913,984): text "Blocked / Low"; alarm colour if FL_DA_PistonSelector4
rectangle at (862,993)-(913,1024): text "Blocked / Low"; alarm colour if FL_A_ExtractCover4
rectangle at (862,1072)-(913,1103): text "Blocked / Low"; alarm colour if RobotGoToInitialPositionBlockedLow
rectangle at (862,1111)-(913,1142): text "Blocked / Low"; alarm colour if RobotGoToPistonHouseBlockedLow
rectangle at (862,1151)-(913,1182): text "Blocked / Low"; alarm colour if RobotGoToSpringHouseBlockedLow
rectangle at (642,1072)-(693,1103): text "Blocked / High"; alarm colour if RobotGoToInitialPositionBlockedHigh
rectangle at (642,1111)-(693,1142): text "Blocked / High"; alarm colour if RobotGoToPistonHouseBlockedHigh
rectangle at (642,1151)-(693,1182): text "Blocked / High"; alarm colour if RobotGoToSpringHouseBlockedHigh
rectangle at (692,1270)-(870,1301): text "----RobotEngine"
rectangle at (862,1270)-(913,1301): text "Blocked / Low"; alarm colour if RobotEngineBlockedLow
rectangle at (689,1190)-(871,1221): text "RobotGoToCoverWarehouse"; alarm colour if F_A_RobotCover4
rectangle at (689,1230)-(871,1261): text "RobotTakeCurrentLoad / ToAssembly"; alarm colour if F_A_RobotAssembly4
rectangle at (863,1190)-(914,1221): text "Blocked / Low"; alarm colour if RobotGoToCoverHouseBlockLow
rectangle at (863,1230)-(914,1261): text "Blocked / Low"; alarm colour if RobotTakeCurrentLoadToAssemblyBlockedLow
rectangle at (643,1190)-(694,1221): text "Blocked / High"; alarm colour if RobotGoToCoverHouseBlockHigh
rectangle at (643,1230)-(694,1261): text "Blocked / High"; alarm colour if RobotTakeCurrentLoadToAssemblyBlockedHigh
12 more shapes without text or variables
*)

(* Visualisation Fault_Simulation
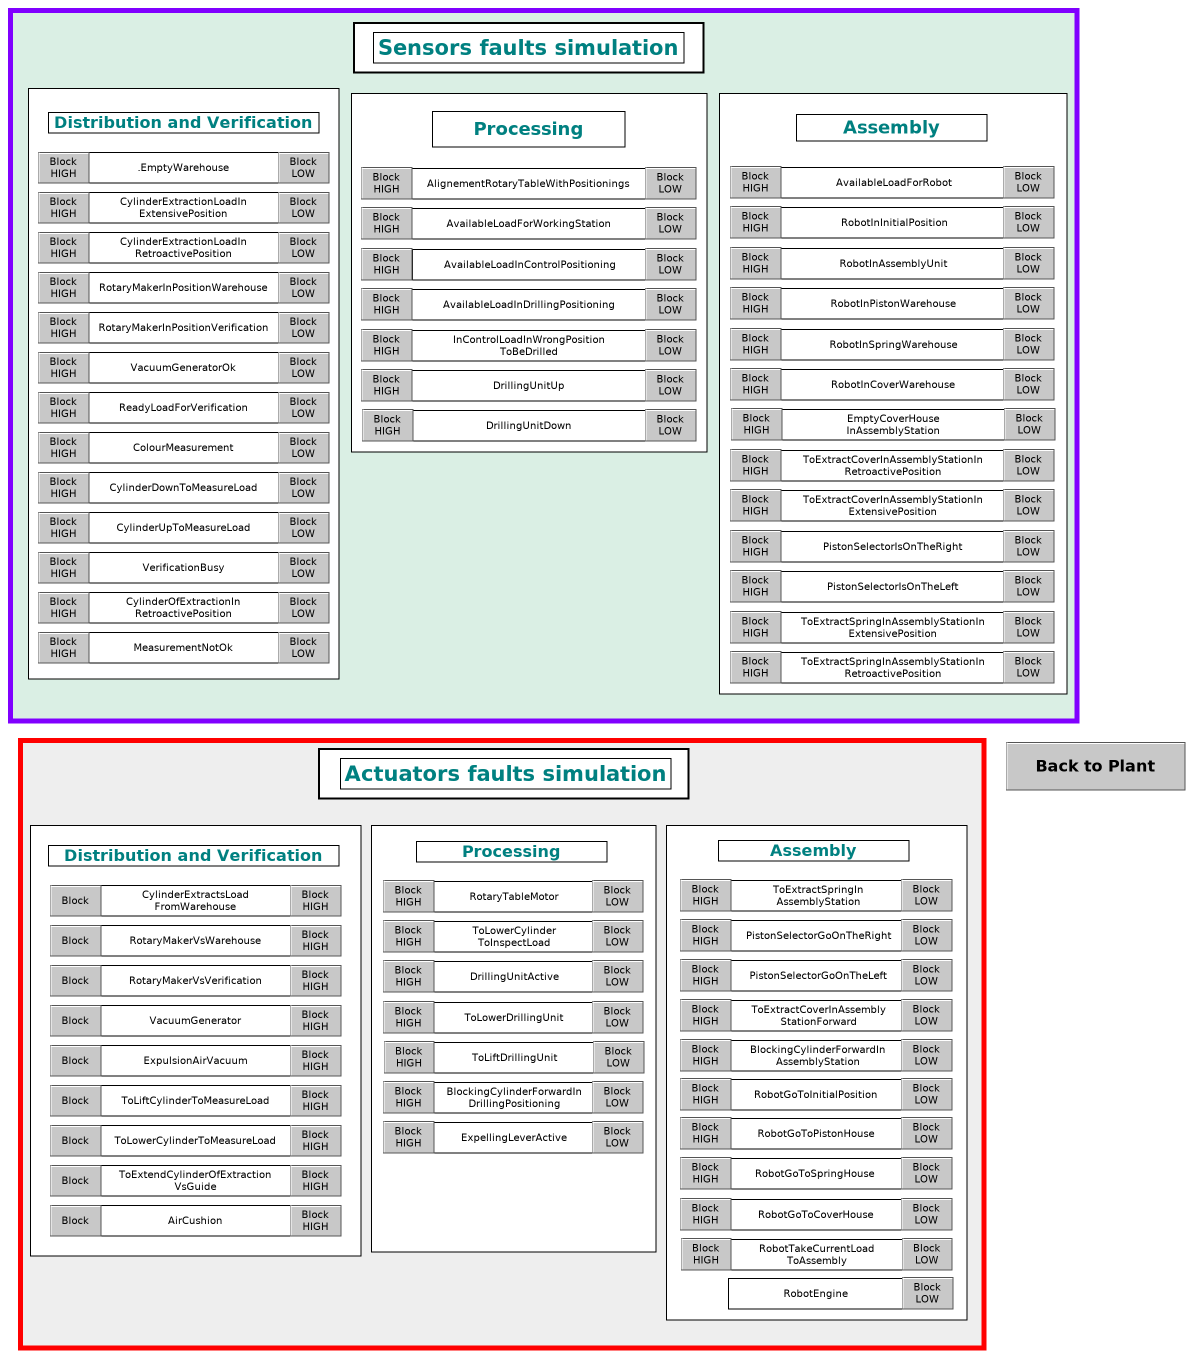
rounded rectangle at (365,34)-(676,65): text "Sensors faults simulation"
rounded rectangle at (332,760)-(663,791): text "Actuators faults simulation"
button at (998,744)-(1177,792): text "Back to Plant"; opens FESTO_Interface
rectangle at (40,114)-(311,135): text "Distribution and Verification"
rectangle at (80,154)-(271,185): text ".EmptyWarehouse"; alarm colour if EmptyWarehouseBlockHigh OR EmptyWarehouseBlockLow
rectangle at (80,194)-(271,225): text "CylinderExtractionLoadIn / ExtensivePosition"; alarm colour if CylinderExtractionLoadInExtensivePositionBlockHigh OR CylinderExtractionLoadInExtensivePositionBlockLow
rectangle at (80,234)-(271,265): text "CylinderExtractionLoadIn / RetroactivePosition"; alarm colour if CylinderExtractionLoadInRetroactivePositionBlockHigh OR CylinderExtractionLoadInRetroactivePositionBlockLow
rectangle at (80,274)-(271,305): text "RotaryMakerInPositionWarehouse"; alarm colour if RotaryMakerInPositionWarehouseBlockHigh OR RotaryMakerInPositionWarehouseBlockLow
rectangle at (80,314)-(271,345): text "RotaryMakerInPositionVerification"; alarm colour if RotaryMakerInPositionVerificationBlockHigh OR RotaryMakerInPositionVerificationBlockLow
rectangle at (80,354)-(271,385): text "VacuumGeneratorOk"; alarm colour if VacuumGeneratorOkBlockHigh OR VacuumGeneratorOkBlockLow
rectangle at (80,394)-(271,425): text "ReadyLoadForVerification"; alarm colour if ReadyLoadForVerificationBlockHigh OR ReadyLoadForVerificationBlockLow
rectangle at (80,434)-(271,465): text "ColourMeasurement"; alarm colour if ColourMeasurementBlockHigh OR ColourMeasurementBlockLow
rectangle at (80,474)-(271,505): text "CylinderDownToMeasureLoad"; alarm colour if CylinderDownToMeasureLoadBlockHigh OR CylinderDownToMeasureLoadBlockLow
rectangle at (80,514)-(271,545): text "CylinderUpToMeasureLoad"; alarm colour if CylinderUpToMeasureLoadBlockHigh OR CylinderUpToMeasureLoadBlockLow
rectangle at (80,554)-(271,585): text "VerificationBusy"; alarm colour if VerificationBusyBlockHigh OR VerificationBusyBlockLow
rectangle at (80,594)-(271,625): text "CylinderOfExtractionIn / RetroactivePosition"; alarm colour if CylinderOfExtractionInRetroactivePositionBlockHigh OR CylinderOfExtractionInRetroactivePositionBlockLow
rectangle at (80,634)-(271,665): text "MeasurementNotOk"; alarm colour if MeasurementNotOkBlockHigh OR MeasurementNotOkBlockLow
button at (30,154)-(81,185): text "Block / HIGH"; toggles EmptyWarehouseBlockHigh
button at (270,154)-(321,185): text "Block / LOW"; toggles EmptyWarehouseBlockLow
button at (30,194)-(81,225): text "Block / HIGH"; toggles CylinderExtractionLoadInExtensivePositionBlockHigh
button at (270,194)-(321,225): text "Block / LOW"; toggles CylinderExtractionLoadInExtensivePositionBlockLow
button at (30,234)-(81,265): text "Block / HIGH"; toggles CylinderExtractionLoadInRetroactivePositionBlockHigh
button at (270,234)-(321,265): text "Block / LOW"; toggles CylinderExtractionLoadInRetroactivePositionBlockLow
button at (30,274)-(81,305): text "Block / HIGH"; toggles RotaryMakerInPositionWarehouseBlockHigh
button at (270,274)-(321,305): text "Block / LOW"; toggles RotaryMakerInPositionWarehouseBlockLow
button at (30,314)-(81,345): text "Block / HIGH"; toggles RotaryMakerInPositionVerificationBlockHigh
button at (270,314)-(321,345): text "Block / LOW"; toggles RotaryMakerInPositionVerificationBlockLow
button at (30,354)-(81,385): text "Block / HIGH"; toggles VacuumGeneratorOkBlockHigh
button at (270,354)-(321,385): text "Block / LOW"; toggles VacuumGeneratorOkBlockLow
button at (30,394)-(81,425): text "Block / HIGH"; toggles ReadyLoadForVerificationBlockHigh
button at (270,394)-(321,425): text "Block / LOW"; toggles ReadyLoadForVerificationBlockLow
button at (30,434)-(81,465): text "Block / HIGH"; toggles ColourMeasurementBlockHigh
button at (270,434)-(321,465): text "Block / LOW"; toggles ColourMeasurementBlockLow
button at (30,474)-(81,505): text "Block / HIGH"; toggles CylinderDownToMeasureLoadBlockHigh
button at (270,474)-(321,505): text "Block / LOW"; toggles CylinderDownToMeasureLoadBlockLow
button at (30,514)-(81,545): text "Block / HIGH"; toggles CylinderUpToMeasureLoadBlockHigh
button at (270,514)-(321,545): text "Block / LOW"; toggles CylinderUpToMeasureLoadBlockLow
button at (30,554)-(81,585): text "Block / HIGH"; toggles VerificationBusyBlockHigh
button at (270,554)-(321,585): text "Block / LOW"; toggles VerificationBusyBlockLow
button at (30,594)-(81,625): text "Block / HIGH"; toggles CylinderOfExtractionInRetroactivePositionBlockHigh
button at (270,594)-(321,625): text "Block / LOW"; toggles CylinderOfExtractionInRetroactivePositionBlockLow
button at (30,634)-(81,665): text "Block / HIGH"; toggles MeasurementNotOkBlockHigh
button at (270,634)-(321,665): text "Block / LOW"; toggles MeasurementNotOkBlockLow
rectangle at (40,847)-(331,868): text "Distribution and Verification"
rectangle at (92,887)-(283,918): text "CylinderExtractsLoad / FromWarehouse"; alarm colour if CylinderExtractsLoadFromWarehouseBlock OR CylinderExtractsLoadFromWarehouseBlockHigh
rectangle at (92,927)-(283,958): text "RotaryMakerVsWarehouse"; alarm colour if RotaryMakerVsWarehouseBlock OR RotaryMakerVsWarehouseBlockHigh
rectangle at (92,967)-(283,998): text "RotaryMakerVsVerification"; alarm colour if RotaryMakerVsVerificationBlock OR RotaryMakerVsVerificationBlockHigh
rectangle at (92,1007)-(283,1038): text "VacuumGenerator"; alarm colour if VacuumGeneratorBlock OR VacuumGeneratorBlockHigh
rectangle at (92,1047)-(283,1078): text "ExpulsionAirVacuum"; alarm colour if ExpulsionAirVacuumBlock OR ExpulsionAirVacuumBlockHigh
rectangle at (92,1087)-(283,1118): text "ToLiftCylinderToMeasureLoad"; alarm colour if ToLiftCylinderToMeasureLoadBlock OR ToLiftCylinderToMeasureLoadBlockHigh
rectangle at (92,1127)-(283,1158): text "ToLowerCylinderToMeasureLoad"; alarm colour if ToLowerCylinderToMeasureLoadBlock OR ToLowerCylinderToMeasureLoadBlockHigh
rectangle at (92,1207)-(283,1238): text "AirCushion"; alarm colour if AirCushionBlock OR AirCushionBlockHigh
rectangle at (92,1167)-(283,1198): text "ToExtendCylinderOfExtraction / VsGuide"; alarm colour if ToExtendCylinderOfExtractionVsGuideBlock OR ToExtendCylinderOfExtractionVsGuideBlockHigh
button at (282,887)-(333,918): text "Block / HIGH"; toggles CylinderExtractsLoadFromWarehouseBlockHigh
button at (282,927)-(333,958): text "Block / HIGH"; toggles RotaryMakerVsWarehouseBlockHigh
button at (282,967)-(333,998): text "Block / HIGH"; toggles RotaryMakerVsVerificationBlockHigh
button at (282,1007)-(333,1038): text "Block / HIGH"; toggles VacuumGeneratorBlockHigh
button at (282,1047)-(333,1078): text "Block / HIGH"; toggles ExpulsionAirVacuumBlockHigh
button at (282,1087)-(333,1118): text "Block / HIGH"; toggles ToLiftCylinderToMeasureLoadBlockHigh
button at (282,1127)-(333,1158): text "Block / HIGH"; toggles ToLowerCylinderToMeasureLoadBlockHigh
button at (282,1167)-(333,1198): text "Block / HIGH"; toggles ToExtendCylinderOfExtractionVsGuideBlockHigh
button at (282,1207)-(333,1238): text "Block / HIGH"; toggles AirCushionBlockHigh
button at (42,887)-(93,918): text "Block"; toggles CylinderExtractsLoadFromWarehouseBlock
button at (42,927)-(93,958): text "Block"; toggles RotaryMakerVsWarehouseBlock
button at (42,967)-(93,998): text "Block"; toggles RotaryMakerVsVerificationBlock
button at (42,1007)-(93,1038): text "Block"; toggles VacuumGeneratorBlock
button at (42,1047)-(93,1078): text "Block"; toggles ExpulsionAirVacuumBlock
button at (42,1087)-(93,1118): text "Block"; toggles ToLiftCylinderToMeasureLoadBlock
button at (42,1127)-(93,1158): text "Block"; toggles ToLowerCylinderToMeasureLoadBlock
button at (42,1167)-(93,1198): text "Block"; toggles ToExtendCylinderOfExtractionVsGuideBlock
button at (42,1207)-(93,1238): text "Block"; toggles AirCushionBlock
rectangle at (424,113)-(617,149): text "Processing"
rectangle at (788,116)-(979,143): text "Assembly"
rectangle at (402,170)-(639,201): text "AlignementRotaryTableWithPositionings"
rectangle at (403,210)-(639,241): text "AvailableLoadForWorkingStation"
rectangle at (404,251)-(640,282): text "AvailableLoadInControlPositioning"
rectangle at (402,291)-(640,322): text "AvailableLoadInDrillingPositioning"
rectangle at (402,332)-(640,363): text "InControlLoadInWrongPosition / ToBeDrilled"
rectangle at (402,372)-(640,403): text "DrillingUnitUp"
rectangle at (403,412)-(639,443): text "DrillingUnitDown"
button at (353,169)-(404,201): text "Block / HIGH"; toggles AlignementRotaryTableWithPositioningsBlockHigh
button at (353,209)-(404,241): text "Block / HIGH"; toggles AvailableLoadForWorkingStationBlockHigh
button at (353,250)-(404,282): text "Block / HIGH"; toggles AvailableLoadInControlPositioningBlockHigh
button at (353,290)-(404,322): text "Block / HIGH"; toggles AvailableLoadInDrillingPositioningBlockHigh
button at (353,331)-(404,363): text "Block / HIGH"; toggles InControlLoadInWrongPositionToBeDrilledBlockHigh
button at (353,371)-(404,403): text "Block / HIGH"; toggles DrillingUnitUpBlockHigh
button at (637,169)-(688,201): text "Block / LOW"; toggles AlignementRotaryTableWithPositioningsBlockLow
button at (637,209)-(688,241): text "Block / LOW"; toggles AvailableLoadForWorkingStationBlockLow
button at (637,250)-(688,282): text "Block / LOW"; toggles AvailableLoadInControlPositioningBlockLow
button at (637,290)-(688,322): text "Block / LOW"; toggles AvailableLoadInDrillingPositioningBlockLow
button at (637,331)-(688,363): text "Block / LOW"; toggles InControlLoadInWrongPositionToBeDrilledBlockLow
button at (637,371)-(688,403): text "Block / LOW"; toggles DrillingUnitUpBlockLow
button at (354,411)-(405,443): text "Block / HIGH"; toggles DrillingUnitDownBlockHigh
button at (637,411)-(688,443): text "Block / LOW"; toggles DrillingUnitDownBlockLow
rectangle at (772,169)-(1000,200): text "AvailableLoadForRobot"
rectangle at (772,209)-(1001,240): text "RobotInInitialPosition"
rectangle at (772,250)-(999,281): text "RobotInAssemblyUnit"
rectangle at (772,290)-(999,321): text "RobotInPistonWarehouse"
rectangle at (772,331)-(999,362): text "RobotInSpringWarehouse"
rectangle at (771,371)-(999,402): text "RobotInCoverWarehouse"
rectangle at (770,411)-(1001,442): text "EmptyCoverHouse / InAssemblyStation"
rectangle at (771,452)-(999,483): text "ToExtractCoverInAssemblyStationIn / RetroactivePosition"
rectangle at (771,492)-(999,523): text "ToExtractCoverInAssemblyStationIn / ExtensivePosition"
rectangle at (770,533)-(1000,564): text "PistonSelectorIsOnTheRight"
rectangle at (770,573)-(1000,604): text "PistonSelectorIsOnTheLeft"
rectangle at (770,614)-(1000,645): text "ToExtractSpringInAssemblyStationIn / ExtensivePosition"
rectangle at (770,654)-(1000,685): text "ToExtractSpringInAssemblyStationIn / RetroactivePosition"
button at (722,168)-(773,200): text "Block / HIGH"; toggles AvailableLoadForRobotBlockHigh
button at (722,208)-(773,240): text "Block / HIGH"; toggles RobotInInitialPositionBlockHigh
button at (722,249)-(773,281): text "Block / HIGH"; toggles RobotInAssemblyUnitBlockHigh
button at (722,289)-(773,321): text "Block / HIGH"; toggles RobotInPistonWarehouseBlockHigh
button at (722,330)-(773,362): text "Block / HIGH"; toggles RobotInSpringWarehouseBlockHigh
button at (722,370)-(773,402): text "Block / HIGH"; toggles RobotInCoverWarehouseBlockHigh
button at (723,410)-(774,442): text "Block / HIGH"; toggles EmptyCoverHouseInAssemblyStationBlockHigh
button at (722,451)-(773,483): text "Block / HIGH"; toggles ToExtractCoverInAssemblyStationInRetroactivePositionBlockHigh
button at (722,491)-(773,523): text "Block / HIGH"; toggles ToExtractCoverInAssemblyStationInExtensivePositionBlockHigh
button at (722,532)-(773,564): text "Block / HIGH"; toggles PistonSelectorIsOnTheRightBlockHigh
button at (722,572)-(773,604): text "Block / HIGH"; toggles PistonSelectorIsOnTheLeftBlockHigh
button at (722,613)-(773,645): text "Block / HIGH"; toggles ToExtractSpringInAssemblyStationInExtensivePositionBlockHigh
button at (722,653)-(773,685): text "Block / HIGH"; toggles ToExtractSpringInAssemblyStationInRetroactivePositionBlockHigh
button at (995,168)-(1046,200): text "Block / LOW"; toggles AvailableLoadForRobotBlockLow
button at (995,208)-(1046,240): text "Block / LOW"; toggles RobotInInitialPositionBlockLow
button at (995,249)-(1046,281): text "Block / LOW"; toggles RobotInAssemblyUnitBlockLow
button at (995,289)-(1046,321): text "Block / LOW"; toggles RobotInPistonWarehouseBlockLow
button at (995,330)-(1046,362): text "Block / LOW"; toggles RobotInSpringWarehouseBlockLow
button at (995,370)-(1046,402): text "Block / LOW"; toggles RobotInCoverWarehouseBlockLow
button at (996,410)-(1047,442): text "Block / LOW"; toggles EmptyCoverHouseInAssemblyStationBlockLow
button at (995,451)-(1046,483): text "Block / LOW"; toggles ToExtractCoverInAssemblyStationInRetroactivePositionBlockLow
button at (995,491)-(1046,523): text "Block / LOW"; toggles ToExtractCoverInAssemblyStationInExtensivePositionBlockLow
button at (995,532)-(1046,564): text "Block / LOW"; toggles PistonSelectorIsOnTheRightBlockLow
button at (995,572)-(1046,604): text "Block / LOW"; toggles PistonSelectorIsOnTheLeftBlockLow
button at (995,613)-(1046,645): text "Block / LOW"; toggles ToExtractSpringInAssemblyStationInExtensivePositionBlockLow
button at (995,653)-(1046,685): text "Block / LOW"; toggles ToExtractSpringInAssemblyStationInRetroactivePositionBlockLow
rectangle at (408,843)-(599,864): text "Processing"
rectangle at (710,842)-(901,863): text "Assembly"
rectangle at (721,882)-(900,913): text "ToExtractSpringIn / AssemblyStation"
rectangle at (722,922)-(900,953): text "PistonSelectorGoOnTheRight"
rectangle at (721,962)-(900,993): text "PistonSelectorGoOnTheLeft"
rectangle at (722,1002)-(900,1033): text "ToExtractCoverInAssembly / StationForward"
rectangle at (720,1042)-(900,1073): text "BlockingCylinderForwardIn / AssemblyStation"
rectangle at (721,1081)-(895,1112): text "RobotGoToInitialPosition"
rectangle at (719,1160)-(895,1191): text "RobotGoToSpringHouse"
rectangle at (721,1120)-(895,1151): text "RobotGoToPistonHouse"
rectangle at (422,883)-(590,914): text "RotaryTableMotor"
rectangle at (423,923)-(590,954): text "ToLowerCylinder / ToInspectLoad"
rectangle at (423,963)-(590,994): text "DrillingUnitActive"
rectangle at (422,1004)-(590,1035): text "ToLowerDrillingUnit"
rectangle at (424,1044)-(590,1075): text "ToLiftDrillingUnit"
rectangle at (422,1124)-(590,1155): text "ExpellingLeverActive"
rectangle at (423,1084)-(590,1115): text "BlockingCylinderForwardIn / DrillingPositioning"
button at (584,882)-(635,914): text "Block / LOW"; toggles RotaryTableMotorBlockLow
button at (584,922)-(635,954): text "Block / LOW"; toggles ToLowerCylinderToInspectLoadBlockLow
button at (584,962)-(635,994): text "Block / LOW"; toggles DrillingUnitActiveBlockLow
button at (584,1003)-(635,1035): text "Block / LOW"; toggles ToLowerDrillingUnitBlockLow
button at (585,1043)-(636,1075): text "Block / LOW"; toggles ToLiftDrillingUnitBlockLow
button at (584,1083)-(635,1115): text "Block / LOW"; toggles BlockingCylinderForwardInDrillingPositioningBlockLow
button at (584,1123)-(635,1155): text "Block / LOW"; toggles ExpellingLeverActiveBlockLow
button at (375,882)-(426,914): text "Block / HIGH"; toggles RotaryTableMotorBlockHigh
button at (375,922)-(426,954): text "Block / HIGH"; toggles ToLowerCylinderToInspectLoadBlockHigh
button at (375,962)-(426,994): text "Block / HIGH"; toggles DrillingUnitActiveBlockHigh
button at (375,1003)-(426,1035): text "Block / HIGH"; toggles ToLowerDrillingUnitBlockHigh
button at (376,1043)-(426,1075): text "Block / HIGH"; toggles ToLiftDrillingUnitBlockHigh
button at (375,1083)-(426,1115): text "Block / HIGH"; toggles BlockingCylinderForwardInDrillingPositioningBlockHigh
button at (375,1123)-(426,1155): text "Block / HIGH"; toggles ExpellingLeverActiveBlockHigh
button at (672,881)-(723,913): text "Block / HIGH"; toggles ToExtractSpringInAssemblyStationBlockHigh
button at (672,921)-(723,953): text "Block / HIGH"; toggles PistonSelectorGoOnTheRightBlockHigh
button at (672,961)-(723,993): text "Block / HIGH"; toggles PistonSelectorGoOnTheLeftBlockHigh
button at (672,1001)-(723,1033): text "Block / HIGH"; toggles ToExtractCoverInAssemblyStationForwardBlockHigh
button at (672,1041)-(723,1073): text "Block / HIGH"; toggles BlockingCylinderForwardInAssemblyStationBlockHigh
button at (672,1080)-(723,1112): text "Block / HIGH"; toggles RobotGoToInitialPositionBlockHigh
button at (672,1119)-(723,1151): text "Block / HIGH"; toggles RobotGoToPistonHouseBlockHigh
button at (672,1159)-(723,1191): text "Block / HIGH"; toggles RobotGoToSpringHouseBlockHigh
button at (893,881)-(944,913): text "Block / LOW"; toggles ToExtractSpringInAssemblyStationBlockLow
button at (893,921)-(944,953): text "Block / LOW"; toggles PistonSelectorGoOnTheRightBlockLow
button at (893,961)-(944,993): text "Block / LOW"; toggles PistonSelectorGoOnTheLeftBlockLow
button at (893,1001)-(944,1033): text "Block / LOW"; toggles ToExtractCoverInAssemblyStationForwardBlockLow
button at (893,1041)-(944,1073): text "Block / LOW"; toggles BlockingCylinderForwardInAssemblyStationBlockLow
button at (893,1080)-(944,1112): text "Block / LOW"; toggles RobotGoToInitialPositionBlockLow
button at (893,1119)-(944,1151): text "Block / LOW"; toggles RobotGoToPistonHouseBlockLow
button at (893,1159)-(944,1191): text "Block / LOW"; toggles RobotGoToSpringHouseBlockLow
rectangle at (720,1280)-(896,1311): text "RobotEngine"
button at (894,1279)-(945,1311): text "Block / LOW"; toggles RobotEngineBlockLow
rectangle at (721,1201)-(895,1232): text "RobotGoToCoverHouse"
rectangle at (721,1241)-(897,1272): text "RobotTakeCurrentLoad / ToAssembly"
button at (672,1200)-(723,1232): text "Block / HIGH"; toggles RobotGoToCoverHouseBlockHigh
button at (673,1240)-(723,1272): text "Block / HIGH"; toggles RobotTakeCurrentLoadToAssemblyBlockHigh
button at (893,1200)-(944,1232): text "Block / LOW"; toggles RobotGoToCoverHouseBlockLow
button at (894,1240)-(944,1272): text "Block / LOW"; toggles RobotTakeCurrentLoadToAssemblyBlockLow
10 more shapes without text or variables
*)

(* Visualisation FESTO_Interface
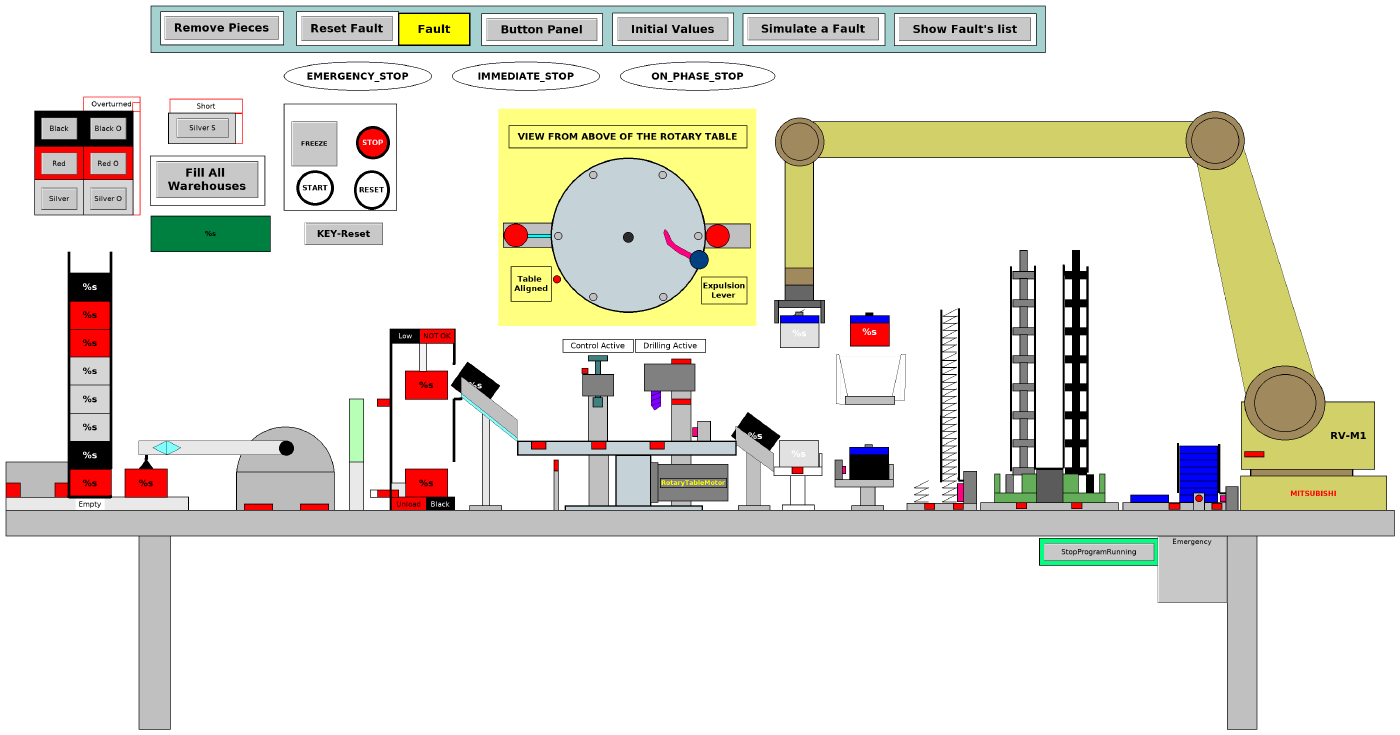
button at (218,82)-(363,134): text "Fill All / Warehouses"; taps FillAllWarehouses
button at (230,-125)-(392,-92): text "Remove Pieces"; taps Remove
button at (425,-125)-(555,-90): text "Reset Fault"; taps FaultDetected
rectangle at (563,-130)-(666,-83): text "Fault"; invisible if NOT PossibleFault
button at (1647,618)-(1746,712): text "Emergency"; toggles NOT EmergencyStop
button at (1062,-123)-(1249,-91): text "Simulate a Fault"; opens Fault_Simulation
button at (1278,-123)-(1466,-90): text "Show Fault's list"; opens Fault_Detection
button at (1485,627)-(1642,652): text "StopProgramRunning"; toggles StopProgramRunning
button at (876,-123)-(1034,-90): text "Initial Values"; opens Initial_Values
rectangle at (583,381)-(614,392): y offset MisuratorPosition
rectangle at (573,381)-(634,422): text "%s"; shows ElementMeasureO; invisible if NOT ElementMeasureBlack OR NOT ElementMeasureCharged; x offset CylinderOfExtractionPosition
rectangle at (573,381)-(634,422): text "%s"; shows ElementMeasureO; invisible if NOT ElementMeasureSilver OR NOT ElementMeasureCharged; x offset CylinderOfExtractionPosition
rectangle at (573,381)-(634,422): text "%s"; shows ElementMeasureO; invisible if NOT ElementMeasureRed OR NOT ElementMeasureCharged; x offset CylinderOfExtractionPosition
rectangle at (5,531)-(94,542): x offset CylinderPosition
rectangle at (83,521)-(94,552): x offset CylinderPosition
rectangle at (493,421)-(514,512): alarm colour if VerificationBusy
rectangle at (533,551)-(554,562): alarm colour if VirtualCylinderDownToMeasureLoad
rectangle at (93,521)-(154,562): text "%s"; shows ElementOneO; invisible if NOT ElementOneBlack OR NOT ElementOneCharged; x offset ElementPosition
rectangle at (93,521)-(154,562): text "%s"; shows ElementOneO; invisible if NOT ElementOneSilver OR NOT ElementOneCharged; x offset ElementPosition
rectangle at (93,521)-(154,562): text "%s"; shows ElementOneO; invisible if NOT ElementOneRed OR NOT ElementOneCharged; x offset ElementPosition
rectangle at (93,481)-(154,522): text "%s"; shows ElementTwoO; invisible if NOT ElementTwoRed OR NOT ElementTwoCharged
rectangle at (93,481)-(154,522): text "%s"; shows ElementTwoO; invisible if NOT ElementTwoSilver OR NOT ElementTwoCharged
rectangle at (93,481)-(154,522): text "%s"; shows ElementTwoO; invisible if NOT ElementTwoBlack OR NOT ElementTwoCharged
rectangle at (93,281)-(154,322): text "%s"; shows ElementSevenO; invisible if NOT ElementSevenSilver OR NOT ElementSevenCharged
rectangle at (93,281)-(154,322): text "%s"; shows ElementSevenO; invisible if NOT ElementSevenBlack OR NOT ElementSevenCharged
rectangle at (93,321)-(154,362): text "%s"; shows ElementSixO; invisible if NOT ElementSixBlack OR NOT ElementSixCharged
rectangle at (93,401)-(154,442): text "%s"; shows ElementFourO; invisible if NOT ElementFourBlack OR NOT ElementFourCharged
rectangle at (93,441)-(154,482): text "%s"; shows ElementThreeO; invisible if NOT ElementThreeBlack OR NOT ElementThreeCharged
rectangle at (93,361)-(154,402): text "%s"; shows ElementFiveO; invisible if NOT ElementFiveBlack OR NOT ElementFiveCharged
rectangle at (93,321)-(154,362): text "%s"; shows ElementSixO; invisible if NOT ElementSixSilver OR NOT ElementSixCharged
rectangle at (93,321)-(154,362): text "%s"; shows ElementSixO; invisible if NOT ElementSixRed OR NOT ElementSixCharged
rectangle at (93,361)-(154,402): text "%s"; shows ElementFiveO; invisible if NOT ElementFiveRed OR NOT ElementFiveCharged
rectangle at (93,401)-(154,442): text "%s"; shows ElementFourO; invisible if NOT ElementFourRed OR NOT ElementFourCharged
rectangle at (93,441)-(154,482): text "%s"; shows ElementThreeO; invisible if NOT ElementThreeRed OR NOT ElementThreeCharged
rectangle at (93,281)-(154,322): text "%s"; shows ElementSevenO; invisible if NOT ElementSevenRed OR NOT ElementSevenCharged
rectangle at (93,441)-(154,482): text "%s"; shows ElementThreeO; invisible if NOT ElementThreeSilver OR NOT ElementThreeCharged
rectangle at (93,361)-(154,402): text "%s"; shows ElementFiveO; invisible if NOT ElementFiveSilver OR NOT ElementFiveCharged
rectangle at (93,401)-(154,442): text "%s"; shows ElementFourO; invisible if NOT ElementFourSilver OR NOT ElementFourCharged
rectangle at (3,541)-(24,562): alarm colour if CylinderExtractionLoadInRetroactivePosition
rectangle at (73,541)-(94,562): alarm colour if CylinderExtractionLoadInExtensivePosition
rectangle at (173,521)-(234,562): text "%s"; shows ElementRotaryO; invisible if NOT ElementRotaryBlack OR NOT ElementRotaryCharged; angle RotaryPosition
rectangle at (173,521)-(234,562): text "%s"; shows ElementRotaryO; invisible if NOT ElementRotaryRed OR NOT ElementRotaryCharged; angle RotaryPosition
rectangle at (173,521)-(234,562): text "%s"; shows ElementRotaryO; invisible if NOT ElementRotarySilver OR NOT ElementRotaryCharged; angle RotaryPosition
rectangle at (114,-10)-(195,11): text "Overturned"
rectangle at (343,571)-(384,582): alarm colour if RotaryMakerInPositionWarehouse
rectangle at (423,571)-(464,582): alarm colour if RotaryMakerInPositionVerification
polygon at (193,481)-(403,501): angle RotaryPosition
rectangle at (237,-7)-(341,14): text "Short"
polygon at (213,481)-(233,501): invisible if NOT ExpulsionAirVacuumVis; angle RotaryPosition
polygon at (233,481)-(253,501): invisible if NOT VacuumGeneratorOk; angle RotaryPosition
rectangle at (533,421)-(554,432): alarm colour if CylinderUpToMeasureLoad
rectangle at (593,341)-(604,382): bottom MisuratorPosition
rectangle at (573,521)-(634,562): text "%s"; shows ElementVerificationO; invisible if NOT ElementVerificationBlack OR NOT ElementVerificationCharged; x offset CylinderOfExtractionPosition; y offset -LiftPosition
rectangle at (573,521)-(634,562): text "%s"; shows ElementVerificationO; invisible if NOT ElementVerificationSilver OR NOT ElementVerificationCharged; x offset CylinderOfExtractionPosition; y offset -LiftPosition
rectangle at (573,521)-(634,562): text "%s"; shows ElementVerificationO; invisible if NOT ElementVerificationRed OR NOT ElementVerificationCharged; x offset CylinderOfExtractionPosition; y offset -LiftPosition
rectangle at (553,541)-(574,562): right CylinderOfExtractionPosition; y offset -LiftPosition
rectangle at (593,561)-(614,582): top -LiftPosition
rectangle at (553,561)-(644,582): y offset -LiftPosition
rectangle at (553,561)-(604,582): text "Load"
rectangle at (553,561)-(604,582): text "Unload"; invisible if ReadyLoadForVerification
rounded rectangle at (593,321)-(644,342): text "Measure"
rounded rectangle at (593,321)-(644,342): text "OK"; invisible if UncorrectComparison OR NOT CylinderUpToMeasureLoad
rectangle at (603,561)-(644,582): text "Bright"; y offset -LiftPosition
rectangle at (603,561)-(644,582): text "Black"; invisible if ColourMeasurement; y offset -LiftPosition
rounded rectangle at (593,321)-(644,342): text "NOT OK"; invisible if NOT UncorrectComparison OR NOT CylinderUpToMeasureLoad
button at (247,21)-(321,48): text "Silver S"; taps Silvershort
button at (54,120)-(105,151): text "Silver"; taps Silver
button at (54,20)-(105,51): text "Black"; taps Black
button at (54,70)-(105,101): text "Red"; taps Red
button at (124,70)-(175,101): text "Red O"; taps Redoverturned
button at (124,120)-(175,151): text "Silver O"; taps Silveroverturned
button at (124,20)-(175,51): text "Black O"; taps Blackoverturned
rectangle at (523,551)-(534,562): alarm colour if CylinderDownToMeasureLoad
rectangle at (173,521)-(234,562): text "%s"; shows ElementWaitingO; invisible if NOT ElementWaitingBlack OR NOT ElementWaitingCharged
rectangle at (173,521)-(234,562): text "%s"; shows ElementWaitingO; invisible if NOT ElementWaitingSilver OR NOT ElementWaitingCharged
rectangle at (173,521)-(234,562): text "%s"; shows ElementWaitingO; invisible if NOT ElementWaitingRed OR NOT ElementWaitingCharged
rectangle at (553,551)-(564,562): alarm colour if CylinderOfExtractionInRetroactivePosition; y offset -LiftPosition
rounded rectangle at (553,321)-(594,342): text "High"
rounded rectangle at (553,321)-(594,342): text "Low"; invisible if MeasurementNotOk
rectangle at (93,241)-(154,282): text "%s"; shows ElementEightO; invisible if NOT ElementEightSilver OR NOT ElementEightCharged
rectangle at (93,241)-(154,282): text "%s"; shows ElementEightO; invisible if NOT ElementEightRed OR NOT ElementEightCharged
rectangle at (93,241)-(154,282): text "%s"; shows ElementEightO; invisible if NOT ElementEightBlack OR NOT ElementEightCharged
rectangle at (103,561)-(144,582): alarm colour if EmptyWarehouse
rectangle at (103,561)-(144,582): text "Empty"; invisible if NOT EmptyWarehouse
button at (689,-122)-(847,-90): text "Button Panel"; opens Switchboard
rectangle at (1773,541)-(1967,577): text "Tesi di Marco Pierantoni / a.a.2007-08"
rounded rectangle at (1564,528)-(1572,565): x offset PistonSelectorPosition
rounded rectangle at (1414,528)-(1422,565): x offset PistonSelectorPosition
rectangle at (901,336)-(1002,355): text "Drilling Active"; invisible if NOT AvailableLoadInDrillingPositioning
polyline at (1223,492)-(1243,522): invisible if NOT SpringAssembly OR SpringNumber<0
polyline at (1123,294)-(1143,324): invisible if NOT SpringInEndEffector OR SpringNumber<0; x offset RobotGoHorizontalPosition; y offset RobotGoVerticalPosition
rectangle at (1736,559)-(1749,568): left -ExtractCoverPosition
rectangle at (1208,305)-(1264,346): text "%s"; shows ElementToDiscardO; invisible if NOT ElementToDiscardSilver OR NOT ElementToDiscard; y offset ElementToDiscardPosition
rectangle at (1208,305)-(1264,346): text "%s"; shows ElementToDiscardO; invisible if NOT ElementToDiscardBlack OR NOT ElementToDiscard; y offset ElementToDiscardPosition
rectangle at (983,462)-(994,475): left BlockingActuator*-1
rectangle at (1115,233)-(1156,288): x offset RobotGoHorizontalPosition; y offset RobotGoVerticalPosition
rectangle at (1191,517)-(1202,528): right CylinderPositionInAssemblyUnit
rectangle at (1137,25)-(1713,77): left RobotGoHorizontalPosition
rounded rectangle at (1766,425)-(1957,522): text "RV-M1"
rectangle at (1361,542)-(1378,568): left -ExtractSpringPosition
rectangle at (1207,501)-(1263,537): invisible if NOT ElementAssemblySilver; angle RotaryPosition*9
rectangle at (1207,501)-(1263,537): invisible if NOT ElementAssemblyRed; angle RotaryPosition*9
rectangle at (1207,500)-(1263,536): invisible if NOT ElementAssemblyBlack; angle RotaryPosition*9
polyline at (1340,387)-(1360,417): invisible if NOT Spring5
polyline at (1340,417)-(1360,447): invisible if NOT Spring4
polyline at (1340,447)-(1360,477): invisible if NOT Spring3
polyline at (1340,324)-(1360,354): invisible if NOT Spring7
polyline at (1340,478)-(1360,508): invisible if NOT Spring2
polyline at (1340,508)-(1360,538): invisible if NOT Spring1
polyline at (1340,356)-(1360,386): invisible if NOT Spring6
rectangle at (1678,498)-(1733,509): invisible if NOT Cover7
rectangle at (1678,508)-(1733,519): invisible if NOT Cover6
rectangle at (1678,518)-(1733,529): invisible if NOT Cover5
rectangle at (1678,528)-(1733,539): invisible if NOT Cover4
rectangle at (1678,538)-(1733,549): invisible if NOT Cover3
rectangle at (1678,548)-(1733,559): invisible if NOT Cover2
rectangle at (1678,558)-(1733,569): invisible if NOT Cover1
rectangle at (1678,488)-(1733,499): invisible if NOT Cover8
rectangle at (1608,558)-(1663,569): invisible if NOT CoverExtract OR CoverNumber<0
rectangle at (1207,490)-(1263,501): invisible if NOT CoverAssembly OR CoverNumber<0
rectangle at (844,361)-(852,430): y offset InspectPosition
rectangle at (1107,480)-(1163,519): text "%s"; shows ElementStation1RobotO; invisible if NOT ElementStation1RobotRed OR NOT ElementStation1RobotCharged
rectangle at (1107,480)-(1163,519): text "%s"; shows ElementStation1RobotO; invisible if NOT ElementStation1RobotBlack OR NOT ElementStation1RobotCharged
rectangle at (1107,480)-(1163,519): text "%s"; shows ElementStation1RobotO; invisible if NOT ElementStation1RobotSilver OR NOT ElementStation1RobotCharged
rectangle at (1125,518)-(1141,528): alarm colour if AvailableLoadForRobot
rectangle at (996,247)-(1061,286): text "Expulsion / Lever"; invisible if NOT ExpellingLeverActive
rectangle at (798,336)-(899,355): text "Control Active"; invisible if NOT AvailableLoadInControlPositioning
rectangle at (721,31)-(1061,63): text "VIEW FROM ABOVE OF THE ROTARY TABLE"
rectangle at (1104,280)-(1167,291): left EndEffectorPosition; right -EndEffectorPosition; x offset RobotGoHorizontalPosition; y offset RobotGoVerticalPosition
rectangle at (1166,280)-(1172,313): x offset (RobotGoHorizontalPosition)-EndEffectorPosition; y offset RobotGoVerticalPosition
rectangle at (1100,280)-(1106,313): x offset (RobotGoHorizontalPosition)+EndEffectorPosition; y offset RobotGoVerticalPosition
rectangle at (1108,307)-(1164,348): text "%s"; shows ElementInEndEffectorO; invisible if NOT ElementInEndEffectorRed OR NOT ElementInEndEffector; x offset RobotGoHorizontalPosition; y offset RobotGoVerticalPosition
rectangle at (1108,307)-(1164,348): text "%s"; shows ElementInEndEffectorO; invisible if NOT ElementInEndEffectorBlack OR NOT ElementInEndEffector; x offset RobotGoHorizontalPosition; y offset RobotGoVerticalPosition
rectangle at (1108,307)-(1164,348): text "%s"; shows ElementInEndEffectorO; invisible if NOT ElementInEndEffectorSilver OR NOT ElementInEndEffector; x offset RobotGoHorizontalPosition; y offset RobotGoVerticalPosition
polygon at (1038,440)-(1108,508): text "%s"; shows ElementAirO; invisible if NOT ElementSleighRed OR NOT ElementSleighCharged; x offset MovementElementSleigh*2; y offset MovementElementSleigh
polygon at (1038,440)-(1108,508): text "%s"; shows ElementAirO; invisible if NOT ElementSleighSilver OR NOT ElementSleighCharged; x offset MovementElementSleigh*2; y offset MovementElementSleigh
polygon at (1038,440)-(1108,508): text "%s"; shows ElementSleighO; invisible if NOT ElementSleighBlack OR NOT ElementSleighCharged; x offset MovementElementSleigh*2; y offset MovementElementSleigh
rounded rectangle at (1765,531)-(1974,582): text "MITSUBISHI"
rectangle at (1115,56)-(1156,243): bottom RobotGoVerticalPosition; x offset RobotGoHorizontalPosition
ellipse at (1101,20)-(1171,89): x offset RobotGoHorizontalPosition
ellipse at (1109,27)-(1163,81): x offset RobotGoHorizontalPosition
polyline at (1341,293)-(1361,323): invisible if NOT Spring8
polyline at (1300,538)-(1320,568): invisible if NOT SpringExtract OR SpringNumber<0
polyline at (1340,538)-(1360,568): invisible if NOT VisualSpring; x offset -ExtractSpringPosition
rectangle at (1663,570)-(1679,579): alarm colour if ToExtractCoverInAssemblyStationInExtensivePosition
rectangle at (1724,570)-(1739,579): alarm colour if ToExtractCoverInAssemblyStationInRetroactivePosition
ellipse at (1701,558)-(1711,568): alarm colour if EmptyCoverHouseInAssemblyStation
rounded rectangle at (1115,234)-(1156,259): x offset RobotGoHorizontalPosition; y offset RobotGoVerticalPosition
rectangle at (953,364)-(981,372): alarm colour if DrillingUnitUp
rectangle at (953,421)-(981,429): alarm colour if DrillingUnitDown
rounded rectangle at (1453,528)-(1534,569): x offset PistonSelectorPosition
rectangle at (1414,555)-(1572,570): x offset PistonSelectorPosition
rectangle at (1524,569)-(1539,578): alarm colour if PistonSelectorIsOnTheRight
rectangle at (1445,569)-(1460,578): alarm colour if PistonSelectorIsOnTheLeft
rectangle at (1355,570)-(1370,579): alarm colour if ToExtractSpringInAssemblyStationInRetroactivePosition
rectangle at (1314,570)-(1329,579): alarm colour if ToExtractSpringInAssemblyStationInExtensivePosition
rectangle at (1108,302)-(1164,313): invisible if NOT CoverInEndEffector OR CoverNumber<0; x offset RobotGoHorizontalPosition; y offset RobotGoVerticalPosition
rectangle at (724,232)-(782,282): text "Table / Aligned"; invisible if NOT AlignementRotaryTableWithPositionings
rectangle at (717,186)-(785,191): invisible if NOT AirCushion
ellipse at (714,171)-(748,204): invisible if NOT ElementAirBlack OR NOT ElementAirCharged; x offset MovementElementAir
ellipse at (714,171)-(748,204): invisible if NOT ElementAirSilver OR NOT ElementAirCharged; x offset MovementElementAir
ellipse at (714,171)-(748,204): invisible if NOT ElementAirRed OR NOT ElementAirCharged; x offset MovementElementAir
ellipse at (1002,172)-(1036,205): invisible if NOT ElementSleighBlack OR NOT ElementSleighCharged; x offset MovementElementSleigh
ellipse at (1002,172)-(1036,205): invisible if NOT ElementSleighSilver OR NOT ElementSleighCharged; x offset MovementElementSleigh
ellipse at (1002,172)-(1036,205): invisible if NOT ElementSleighRed OR NOT ElementSleighCharged; x offset MovementElementSleigh
rectangle at (841,419)-(855,433): y offset InspectPosition
rectangle at (834,359)-(862,367): y offset InspectPosition
rectangle at (1208,305)-(1264,346): text "%s"; shows ElementToDiscardO; invisible if NOT ElementToDiscardRed OR NOT ElementToDiscard; y offset ElementToDiscardPosition
rectangle at (1208,302)-(1264,313): invisible if NOT CoverToDiscard OR CoverNumber<0; y offset ElementToDiscardPosition
rectangle at (1194,360)-(1280,421): text "%s"; shows CanText; invisible if NOT CanDiscard; alarm colour if CanColour
polygon at (1188,357)-(1207,429): invisible if NOT CanDiscard
polygon at (1267,357)-(1287,423): invisible if NOT CanDiscard
rectangle at (1201,417)-(1272,429): invisible if NOT CanDiscard
rectangle at (825,377)-(834,385): alarm colour if InControlLoadInWrongPositionToBeDrilled
rectangle at (1771,496)-(1799,504): alarm colour if LightRobotInMovement
rectangle at (914,371)-(987,410): y offset DrillingUnitPosition/2
ellipse at (784,245)-(795,256): alarm colour if AlignementRotaryTableWithPositionings
ellipse at (786,183)-(797,194): angle RotaryTableVisual
ellipse at (836,96)-(847,107): angle RotaryTableVisual
ellipse at (986,183)-(997,194): angle RotaryTableVisual
ellipse at (935,96)-(946,107): angle RotaryTableVisual
ellipse at (936,270)-(947,281): angle RotaryTableVisual
ellipse at (836,270)-(847,281): angle RotaryTableVisual
polygon at (942,180)-(993,228): angle LeverPosition
rectangle at (753,482)-(774,493): alarm colour if AvailableLoadForWorkingStation
rectangle at (839,482)-(860,493): alarm colour if AvailableLoadInControlPositioning
rectangle at (922,482)-(943,493): alarm colour if AvailableLoadInDrillingPositioning
rounded rectangle at (923,512)-(934,569): alarm colour if RotaryTableMotor
rectangle at (937,534)-(1032,548): text "RotaryTableMotor"; invisible if NOT RotaryTableMotor
rectangle at (785,508)-(792,524): alarm colour if AlignementRotaryTableWithPositionings
ellipse at (503,32)-(551,79): text "STOP"; taps Stop
ellipse at (500,95)-(551,151): text "RESET"; alarm colour if LightReset; taps Reset
ellipse at (418,95)-(471,145): text "START"; alarm colour if LightStart; taps Start
button at (411,25)-(476,89): text "FREEZE"; toggles NOT FreezeStopPuls
polygon at (638,368)-(708,436): text "%s"; shows ElementAirO; invisible if NOT ElementAirRed OR NOT ElementAirCharged; x offset MovementElementAir*2; y offset MovementElementAir
polygon at (638,368)-(708,436): text "%s"; shows ElementAirO; invisible if NOT ElementAirSilver OR NOT ElementAirCharged; x offset MovementElementAir*2; y offset MovementElementAir
polygon at (638,368)-(708,436): text "%s"; shows ElementAirO; invisible if NOT ElementAirBlack OR NOT ElementAirCharged; x offset MovementElementAir*2; y offset MovementElementAir
polygon at (653,413)-(733,482): invisible if NOT AirCushion
ellipse at (400,-60)-(611,-19): text "EMERGENCY_STOP"; alarm colour if EmergencyInStop
ellipse at (640,-60)-(851,-19): text "IMMEDIATE_STOP"; alarm colour if ImmediateInStop
ellipse at (880,-60)-(1101,-19): text "ON_PHASE_STOP"; alarm colour if OnPhaseInStop
button at (430,170)-(541,201): text "KEY-Reset"; taps KeyReset
rectangle at (210,160)-(381,211): text "%s"; shows TextMachineEmptyForReset; invisible if ButtonMachineToBeEmptyInvisible; alarm colour if LightMachineToBeEmpty; toggles MachineNOTOkForReset
157 more shapes without text or variables
12 elements of other kinds (tables, trends, ...) not read
*)

(* Visualisation Initial_Values
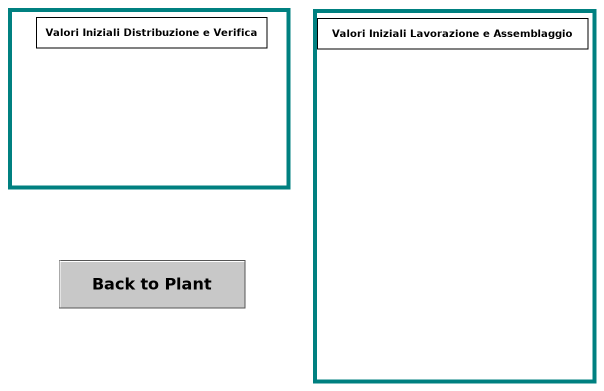
rectangle at (51,28)-(282,59): text "Valori Iniziali Distribuzione e Verifica"
rectangle at (332,29)-(603,60): text "Valori Iniziali Lavorazione e Assemblaggio"
button at (74,271)-(260,319): text "Back to Plant"; opens FESTO_Interface
2 more shapes without text or variables
7 elements of other kinds (tables, trends, ...) not read
*)

(* Visualisation Switchboard
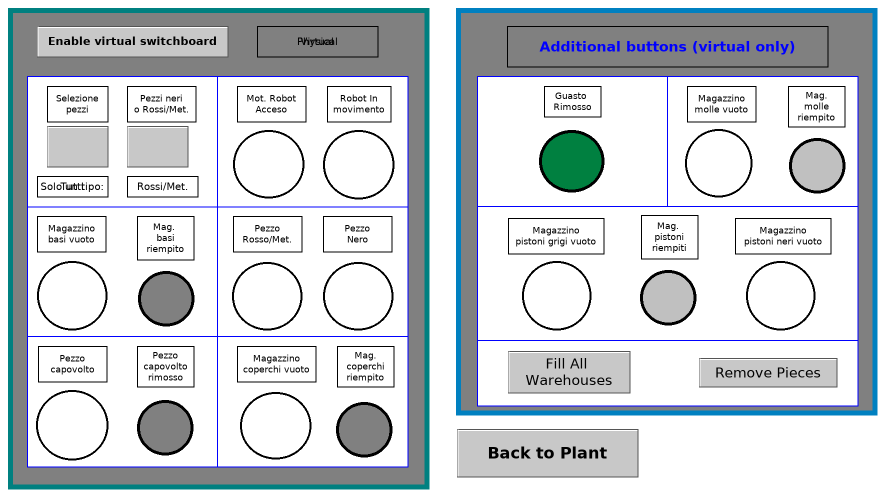
rectangle at (557,100)-(614,131): text "Guasto / Rimosso"
ellipse at (151,285)-(207,340): taps FullWarehousePuls
ellipse at (349,416)-(405,471): taps CoverLoad
rectangle at (801,100)-(858,141): text "Mag. / molle / riempito"
rectangle at (150,230)-(207,274): text "Mag. / basi / riempito"; alarm colour if FullWarehousePuls
rectangle at (350,360)-(407,401): text "Mag. / coperchi / riempito"; alarm colour if FullWareHouseInAssemblyStationPuls
rectangle at (700,100)-(769,136): text "Magazzino / molle vuoto"
rectangle at (50,230)-(119,266): text "Magazzino / basi vuoto"
rectangle at (250,360)-(329,396): text "Magazzino / coperchi vuoto"
rectangle at (51,360)-(120,396): text "Pezzo / capovolto"
rectangle at (246,230)-(315,266): text "Pezzo / Rosso/Met."
rectangle at (336,230)-(405,266): text "Pezzo / Nero"
rectangle at (250,100)-(319,136): text "Mot. Robot / Acceso"
rectangle at (340,100)-(404,136): text "Robot In / movimento"
ellipse at (150,414)-(206,469): taps UpsideDownLoadRemovedInExpellingPuls
rectangle at (150,360)-(207,401): text "Pezzo / capovolto / rimosso"; alarm colour if UpsideDownLoadRemovedInExpellingPuls
rectangle at (140,100)-(209,136): text "Pezzi neri / o Rossi/Met."
button at (60,140)-(121,181): toggles ToWorkBlackOrRedLoad
button at (140,140)-(201,181): toggles ToWorkBlackLoadPuls
rounded rectangle at (520,40)-(841,81): text "Additional buttons (virtual only)"
rounded rectangle at (50,190)-(121,211): text "Tutti"; invisible if NOT ToWorkBlackOrRedLoad
rounded rectangle at (140,190)-(211,211): text "Neri"; invisible if NOT ToWorkBlackLoad
rounded rectangle at (140,190)-(211,211): text "Rossi/Met."; invisible if ToWorkBlackLoad
button at (50,40)-(241,71): text "Enable virtual switchboard"; toggles EnableVirtualBox
rectangle at (270,40)-(391,71): text "Virtual"
rectangle at (270,40)-(391,71): text "Physical"; invisible if EnableVirtualBox
rounded rectangle at (50,190)-(121,211): text "Solo un tipo:"; invisible if ToWorkBlackOrRedLoad
rectangle at (60,100)-(121,136): text "Selezione / pezzi"
ellipse at (535,275)-(604,344): alarm colour if EmptyPistonSilverWarehouse
rectangle at (654,229)-(711,273): text "Mag. / pistoni / riempiti"
rectangle at (521,232)-(617,268): text "Magazzino / pistoni grigi vuoto"
ellipse at (653,284)-(709,339): taps PistonLoad
ellipse at (759,275)-(828,344): alarm colour if EmptyPistonBlackWarehouse
rectangle at (748,232)-(844,268): text "Magazzino / pistoni neri vuoto"
ellipse at (552,144)-(617,206): taps FaultDetected
ellipse at (698,143)-(765,211): alarm colour if EmptySpringWarehouse
ellipse at (336,144)-(407,213): alarm colour if LightRobotInMovement
ellipse at (246,144)-(317,212): alarm colour if LightRobotServoON
ellipse at (802,152)-(858,207): taps SpringLoad
ellipse at (245,276)-(315,344): alarm colour if LightRedLoad
ellipse at (336,276)-(406,344): alarm colour if LightBlackLoad
ellipse at (50,275)-(120,344): alarm colour if LightEmptyWarehouse
ellipse at (49,404)-(121,474): alarm colour if LightUpsideDownLoadInExpelling
ellipse at (253,406)-(324,473): alarm colour if EmptyCoverHouseInAssemblyStation
button at (470,443)-(651,491): text "Back to Plant"; opens FESTO_Interface
button at (521,365)-(643,407): text "Fill All / Warehouses"; taps FillAllWarehouses
button at (712,372)-(850,401): text "Remove Pieces"; taps Remove
12 more shapes without text or variables
*)

(* Visualisation Virtual_Panel
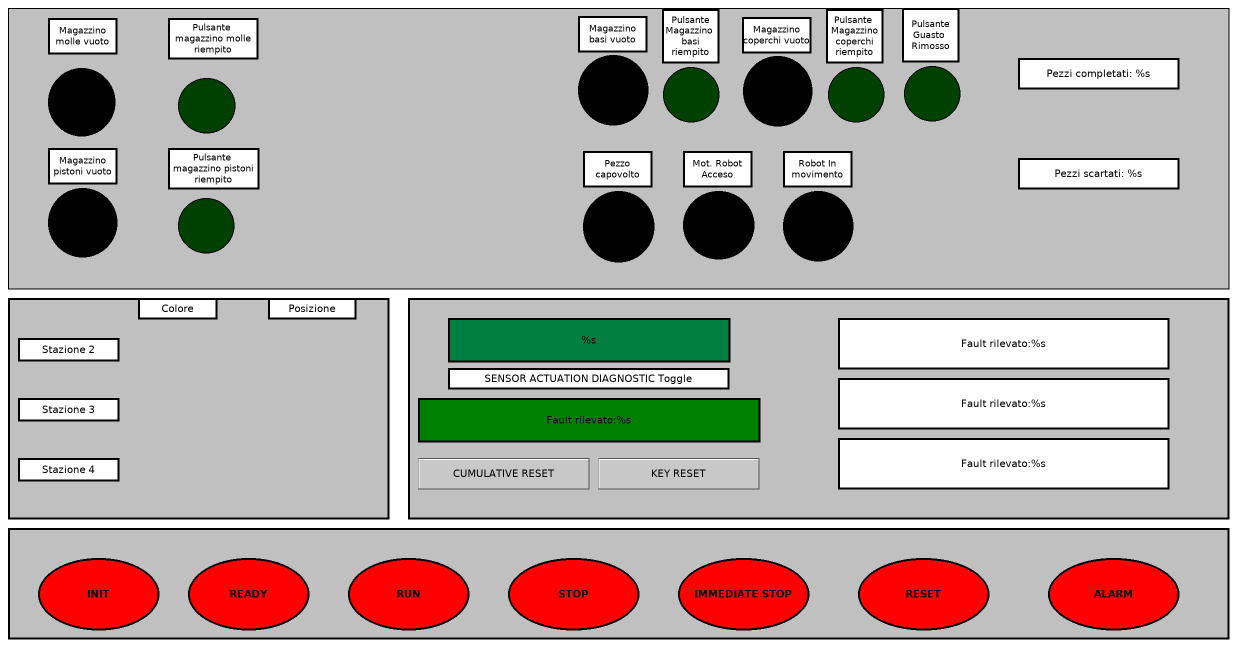
ellipse at (70,70)-(137,138): alarm colour if NOT SpringHouseNotEmpty
ellipse at (70,190)-(139,259): alarm colour if NOT PistonHouseNotEmpty
ellipse at (200,80)-(257,135): taps B_SpringLoader
ellipse at (200,200)-(256,255): taps B_PistonLoader
ellipse at (600,57)-(670,127): alarm colour if LightEmptyWarehouse
ellipse at (605,193)-(676,264): alarm colour if LightUpsideDownLoadInExpelling
ellipse at (765,58)-(834,128): alarm colour if LightEmptyCoverHouse
ellipse at (685,69)-(741,124): taps FullWarehousePuls
ellipse at (850,69)-(906,124): taps CoverLoad
rectangle at (40,400)-(141,423): text "Stazione 3"
rectangle at (190,20)-(280,61): text "Pulsante / magazzino molle / riempito"
rectangle at (684,11)-(741,65): text "Pulsante / Magazzino / basi / riempito"
rectangle at (848,11)-(905,65): text "Pulsante / Magazzino / coperchi / riempito"
rectangle at (70,20)-(139,56): text "Magazzino / molle vuoto"
rectangle at (70,150)-(139,186): text "Magazzino / pistoni vuoto"
rectangle at (600,18)-(669,54): text "Magazzino / basi vuoto"
rectangle at (764,19)-(833,55): text "Magazzino / coperchi vuoto"
rectangle at (605,153)-(674,189): text "Pezzo / capovolto"
ellipse at (805,193)-(875,263): alarm colour if LightRobotInMovement
rectangle at (705,153)-(774,189): text "Mot. Robot / Acceso"
rectangle at (805,153)-(874,189): text "Robot In / movimento"
ellipse at (705,193)-(776,261): alarm colour if LightRobotServoON
ellipse at (60,560)-(181,632): text "INIT"; alarm colour if IndicatorStateInit
ellipse at (1070,560)-(1201,632): text "ALARM"; alarm colour if IndicatorStateAlarm
ellipse at (210,560)-(331,632): text "READY"; alarm colour if IndicatorStateReady
ellipse at (370,560)-(491,632): text "RUN"; alarm colour if IndicatorStateRun
ellipse at (530,560)-(661,632): text "STOP"; alarm colour if IndicatorStateStop
ellipse at (700,560)-(831,632): text "IMMEDIATE STOP"; alarm colour if IndicatorStateFreeze
ellipse at (926,68)-(982,123): taps FaultDetected
rectangle at (924,10)-(981,64): text "Pulsante / Guasto / Rimosso"
rectangle at (440,400)-(782,444): text "Fault rilevato:%s"; shows TypeOfFault; alarm colour if FaultDetected OR PossibleFault; taps FaultRemoved
ellipse at (880,560)-(1011,632): text "RESET"; alarm colour if IndicatorStateReset
button at (440,460)-(611,491): text "CUMULATIVE RESET"; toggles CumulativeReset
button at (620,460)-(781,491): text "KEY RESET"; taps KeyReset
rectangle at (40,460)-(141,483): text "Stazione 4"
rectangle at (1040,60)-(1201,91): text "Pezzi completati: %s"; shows ElementCompleted4
rectangle at (1040,160)-(1201,191): text "Pezzi scartati: %s"; shows ElementRejected4
rectangle at (860,320)-(1191,371): text "Fault rilevato:%s"; shows TypeOfFault1
rectangle at (860,380)-(1191,431): text "Fault rilevato:%s"; shows TypeOfFault2
rectangle at (860,440)-(1191,491): text "Fault rilevato:%s"; shows TypeOfFault3
rectangle at (470,320)-(752,364): text "%s"; shows TextMachineEmptyForReset; invisible if ButtonMachineToBeEmptyInvisible; alarm colour if LightMachineToBeEmpty; toggles MachineNOTOkForReset
rectangle at (470,370)-(751,391): text "SENSOR ACTUATION DIAGNOSTIC Toggle"; alarm colour if SensorActuationDiagnosticEnabled; toggles SensorActuationDiagnosticEnabled
rectangle at (160,300)-(239,321): text "Colore"
rectangle at (40,340)-(141,363): text "Stazione 2"
rectangle at (290,300)-(378,321): text "Posizione"
rectangle at (190,150)-(281,191): text "Pulsante / magazzino pistoni / riempito"
4 more shapes without text or variables
7 elements of other kinds (tables, trends, ...) not read
*)
